// TwinCAT 3 PLC project TcoTixonFeeding
// Title: TcoTixonFeeding
// Company: Vortex.Library
// Author: TcOpenGroup
// ProjectVersion: 0.6.0.913
// ProgramVersion: 3.1.4024.12
// libraries:
//   Tc2_Standard, * (Beckhoff Automation GmbH)
//   Tc2_System, * (Beckhoff Automation GmbH)
//   Tc3_Module, * (Beckhoff Automation GmbH)
//   TcoAbstractions, 0.6.0.913 (Vortex.Library)
//   TcoCore, 0.6.0.913 (Vortex.Library)
//   TcoIo, 0.6.0.913 (Vortex.Library)
//   TcoUtilities, 0.6.0.913 (Vortex.Library)
// project tree:
//   DUTs/ TcoTixonGenericConfig.TcDUT, TcoTixonGenericPickConfig.TcDUT, TcoTixonGenericControl.TcDUT, TcoTixonGenericStatus.TcDUT
//   DUTs/TixonPickStep/ TcoTixonPickStep_Config_v_1_x_x.TcDUT, TcoTixonPickStep_Control_v_1_x_x.TcDUT, TcoTixonPickStep_Status_v_1_x_x.TcDUT
//   DUTs/TixonPickVibroBasic/ TcoTixonPickVibroBasic_Config_v_1_x_x.TcDUT, TcoTixonPickVibroBasic_Control_v_1_x_x.TcDUT, TcoTixonPickVibroBasic_Status_v_1_x_x.TcDUT
//   DUTs/TixonStep/ TcoTixonStep_Config_v_1_x_x.TcDUT, TcoTixonStep_Control_v_1_x_x.TcDUT, TcoTixonStep_Status_v_1_x_x.TcDUT
//   DUTs/TixonVibro/ TcoTixonVibro_Config_v_1_x_x.TcDUT, TcoTixonVibro_Control_v_1_x_x.TcDUT, TcoTixonVibro_Status_v_1_x_x.TcDUT
//   DUTs/TixonPickVibro/ TcoTixonPickVibro_Config_v_1_x_x.TcDUT, TcoTixonPickVibro_Control_v_1_x_x.TcDUT, TcoTixonPickVibro_Status_v_1_x_x.TcDUT
//   / PlcTask.TcTTO
//   POUs/ MAIN.TcPOU
//   POUs/Prototypes/GenericTasks/Base/ TcoTixonFeedingTask.TcPOU
//   POUs/Prototypes/GenericTasks/Buffer/ TcoTixonBufferTask.TcPOU, TcoTixonPickBufferTask.TcPOU
//   POUs/Prototypes/GenericTasks/Hopper/ TcoTixonHopperTask.TcPOU
//   POUs/Prototypes/TiconPickStep/Taks/Step/ TcoTixonPickStepTask.TcPOU
//   POUs/Prototypes/TiconPickStep/Taks/ TcoTixonPickStepSeparatorTask.TcPOU
//   POUs/Prototypes/TiconPickStep/ TcoTixonPickStep_v_1_x_x.TcPOU
//   POUs/Prototypes/TiconPickVibro/Taks/ TcoTixonPickVibroFeederTask.TcPOU, TcoTixonPickVibroSeparatorTask.TcPOU
//   POUs/Prototypes/TiconPickVibro/ TcoTixonPickVibro_v_1_x_x.TcPOU
//   POUs/Prototypes/TixonPickVibroBasic/Tasks/ TcoTixonPickVibroBasicSeparatorTask.TcPOU
//   POUs/Prototypes/TixonPickVibroBasic/ TcoTixonPickVibroBasic_v_1_x_x.TcPOU
//   POUs/Prototypes/TixonStep/Tasks/Separe/ TcoTixonStepSeparatorTask.TcPOU
//   POUs/Prototypes/TixonStep/Tasks/Step/ TcoTixonStepTask.TcPOU
//   POUs/Prototypes/TixonStep/ TcoTixonStep_v_1_x_x.TcPOU
//   POUs/Prototypes/TixonVibro/Tasks/Separe/ TcoTixonVibroSeparatorTask.TcPOU
//   POUs/Prototypes/TixonVibro/ TcoTixonVibro_v_1_x_x.TcPOU
// real-time tasks:
//   TASK PlcTask: cycle T#10ms, priority 20, ADS port 350
//   TASK PlcTask1: cycle T#10ms, priority 1, ADS port 351
//   TASK PN: cycle T#8ms, priority 2, ADS port 301
// I/O:
//   DEVICE Device 4 (EtherCAT) (disabled), AmsNetId 172.20.10.104.5.1
//     Term 1 (EK1100) [EK1100 EtherCAT Coupler (2A E-Bus)]
//       Term 2 (EL1008) [EL1008 8Ch. Dig. Input 24V, 3ms]
//       Term 3 (EL2008) [EL2008 8Ch. Dig. Output 24V, 0.5A]
//       Term 4 (EL3052) [EL3052 2Ch. Ana. Input 4-20mA]
//       Term 5 (EL9576) [EL9576 Brake chopper terminal]
//       Term 6 (EL7211-0010) [EL7211-0010 1Ch. MDP742 Servo motor output stage with OCT (50V, 4.5A RMS)]
//       Term 14 (EL7047) [EL7047 1Ch. Stepper motor output stage (50V, 5A)]
//       Term 8 (EL9011) [EL9011 End Terminal]
//   DEVICE Device 1 (EtherCAT) (disabled), AmsNetId 192.168.4.1.2.1
//     Drive 7 (IndraDrive MPB20) [IndraDrive MPB20]
//   DEVICE ECAT (disabled), AmsNetId 192.168.4.1.3.1
//     EK1200 [EK1200-5000 EtherCAT Power supply (2A E-Bus)]
//       IA1 [EL1008 8Ch. Dig. Input 24V, 3ms]
//       QA1 [EL2008 8Ch. Dig. Output 24V, 0.5A]
//       Term 4 (EL9011) [EL9011 End Terminal]
// variable links:
//   TcoTixonFeedingTests/TcoTixonFeedingTests Instance <-> ECAT
//     PlcTask1 Inputs/GVL_iXlinker.ECAT_x.InfoData.AmsNetId <-> InfoData/AmsNetId
//     PlcTask1 Inputs/GVL_iXlinker.ECAT_x.InfoData.CfgSlaveCount <-> InfoData/CfgSlaveCount
//     PlcTask1 Inputs/GVL_iXlinker.ECAT_x.InfoData.ChangeCount <-> InfoData/ChangeCount
//     PlcTask1 Inputs/GVL_iXlinker.ECAT_x.InfoData.DevId <-> InfoData/DevId
//     PlcTask1 Inputs/GVL_iXlinker.ECAT_x.Inputs.DevState <-> Inputs/DevState
//     PlcTask1 Inputs/GVL_iXlinker.ECAT_x.Inputs.Frm0InputToggle <-> Inputs/Frm0InputToggle
//     PlcTask1 Inputs/GVL_iXlinker.ECAT_x.Inputs.Frm0State <-> Inputs/Frm0State
//     PlcTask1 Inputs/GVL_iXlinker.ECAT_x.Inputs.Frm0WcState <-> Inputs/Frm0WcState
//     PlcTask1 Inputs/GVL_iXlinker.ECAT_x.Inputs.SlaveCount <-> Inputs/SlaveCount
//     PlcTask1 Outputs/GVL_iXlinker.ECAT_x.Outputs.DevCtrl <-> Outputs/DevCtrl
//     PlcTask1 Outputs/GVL_iXlinker.ECAT_x.Outputs.Frm0Ctrl <-> Outputs/Frm0Ctrl
//     PlcTask1 Outputs/GVL_iXlinker.ECAT_x.Outputs.Frm0WcCtrl <-> Outputs/Frm0WcCtrl
//   TcoTixonFeedingTests/TcoTixonFeedingTests Instance <-> ECAT/EK1200/IA1
//     PlcTask1 Inputs/GVL_iXlinker.ECAT_x.EK1200.IA1.Channel_{1..8}.Input <-> Channel {1..8}/Input  (8 links)
//     PlcTask1 Inputs/GVL_iXlinker.ECAT_x.EK1200.IA1.InfoData.State <-> InfoData/State
//     PlcTask1 Inputs/GVL_iXlinker.ECAT_x.EK1200.IA1.WcState.InputToggle <-> WcState/InputToggle
//     PlcTask1 Inputs/GVL_iXlinker.ECAT_x.EK1200.IA1.WcState.WcState <-> WcState/WcState
//   TcoTixonFeedingTests/TcoTixonFeedingTests Instance <-> ECAT/EK1200/QA1
//     PlcTask1 Inputs/GVL_iXlinker.ECAT_x.EK1200.QA1.InfoData.State <-> InfoData/State
//     PlcTask1 Inputs/GVL_iXlinker.ECAT_x.EK1200.QA1.WcState.WcState <-> WcState/WcState
//     PlcTask1 Outputs/GVL_iXlinker.ECAT_x.EK1200.QA1.Channel_{1..8}.Output <-> Channel {1..8}/Output  (8 links)

CONFIGURATION TcoTixonFeeding
    RESOURCE PLC ON TwinCAT3
        TASK PlcTask(INTERVAL := T#10ms, PRIORITY := 20);
        PROGRAM MAIN WITH PlcTask : MAIN;
    END_RESOURCE
END_CONFIGURATION

// ---- DUTs/TcoTixonGenericConfig.TcDUT
TYPE TcoTixonGenericConfig :
STRUCT
    {attribute addProperty Name "<#Blink period#> - T_BLINK"}
    BlinkTime : TIME := T#500MS;
    {attribute addProperty Name "<#Feeder empty time to report#> - T_SIG_EMPTY"}
    FeederEmptyTime : TIME := T#5S;
    {attribute addProperty Name "<#Buffer empty time to report#> - T_BUF_EMPTY"}
    BufferEmptyTime : TIME := T#1S;
    {attribute addProperty Name "<#Buffer full time to report#> - T_BUF_FULL"}
    BufferFullTime : TIME := T#1S;
    {attribute addProperty Name "<#Buffer blow on start#> - T_BUF_BLOW_ON"}
    BufferBlowStartTime : TIME := T#300MS;
    {attribute addProperty Name "<#Buffer time to idle#> - T_BUF_IDLE"}
    BufferIdleTime : TIME := T#5S;
    {attribute addProperty Name "<#Buffer full blow time after#> - T_BUF_BLOW_FULL"}
    BufferBlowFullTime : TIME := T#1S;
    {attribute addProperty Name "<#Buffer blow  active #>"}
    BufferBlowActive : BOOL := TRUE;
    {attribute addProperty Name "<#Time when component in separator #> - T_BUFSEP_ON"}
    TimeToComponentInSeparator : TIME := T#300MS;
    {attribute addProperty Name "<#Time when component is out of separator #> - T_FLY_OFF"}
    TimeToComponentOutSeparator : TIME := T#1S;
    {attribute addProperty Name "<#Hooper is active#>"}
    HopperActive : BOOL := FALSE;
    {attribute addProperty Name "<#Time to hopper start #> - T_HOOP_ON"}
    TimeToHopperStart : TIME := T#5S;
    {attribute addProperty Name "<#Time to hopper run #> - T_HOOP_RUN"}
    TimeToHopperRun : TIME := T#30S;
END_STRUCT
END_TYPE

// ---- DUTs/TcoTixonGenericPickConfig.TcDUT
TYPE TcoTixonGenericPickConfig EXTENDS TcoTixonGenericConfig :
STRUCT
    {attribute addProperty Name "<#Separator  active #>"}
    SeparatorActive : BOOL := TRUE;
END_STRUCT
END_TYPE

// ---- DUTs/TcoTixonGenericControl.TcDUT
TYPE TcoTixonGenericControl :
STRUCT
    {attribute addProperty Name "<#Feeding A #> - q1"}
    FeedingA : BOOL;
    {attribute addProperty Name "<#Separe component#> - q2"}
    SepareComponent : BOOL;
    {attribute addProperty Name "<#Blow A#> - q3"}
    BlowAValve : BOOL;
    {attribute addProperty Name "<#Red led#> - q4"}
    RedLed : BOOL;
    {attribute addProperty Name "<#Green led#> - q5"}
    GreenLed : BOOL;
    {attribute addProperty Name "<#Hooper#> - q6"}
    Hooper : BOOL;
END_STRUCT
END_TYPE

// ---- DUTs/TcoTixonGenericStatus.TcDUT
TYPE TcoTixonGenericStatus :
STRUCT
    ActionDescription : STRING(100);
    {attribute addProperty Name "<#Component is ready#>"}
    ComponentReady : BOOL;
    {attribute addProperty Name "<#Tixon controller in auto#> - i1"}
    ControllerInAuto : BOOL;
    {attribute addProperty Name "<#Feeder has components#> - i2"}
    NotEmptyFeeder : BOOL;
    {attribute addProperty Name "<#Separator in home position#> - i3"}
    SeparatorHomePos : BOOL;
    {attribute addProperty Name "<#Filing sensor#> - i4"}
    FillingSensor : BOOL;
    {attribute addProperty Name "<#Separator present#> - i5"}
    SeparatorPresent : BOOL;
END_STRUCT
END_TYPE

// ---- DUTs/TixonPickStep/TcoTixonPickStep_Config_v_1_x_x.TcDUT
TYPE TcoTixonPickStep_Config_v_1_x_x EXTENDS TcoTixonGenericPickConfig :
STRUCT
    {attribute addProperty Name "<#Time when stepper in work #> - T_STEP_WORK"}
    SteperInWorkTime : TIME := T#1S;
    {attribute addProperty Name "<#Time when stepper in home #> - T_STEP_HOME"}
    SteperInHomeTime : TIME := T#1S;
    {attribute addProperty Name "<#Error time separator #> - T_SEP_ERROR"}
    ErrorTimeSeparator : TIME := T#0S;
    {attribute addProperty Name "<#Error time buffer #> - T_BUFF_ERROR"}
    ErrorTimeBuffer : TIME := T#0S;
    {attribute addProperty Name "<#Error time Stepper #> - T_STEP_ERROR"}
    ErrorTimeStepper : TIME := T#0S;
    {attribute addProperty Name "<#Error time Hopper #> - T_HOP_ERROR"}
    ErrorTimeHopper : TIME := T#0S;
END_STRUCT
END_TYPE

// ---- DUTs/TixonPickStep/TcoTixonPickStep_Control_v_1_x_x.TcDUT
TYPE TcoTixonPickStep_Control_v_1_x_x EXTENDS TcoTixonGenericControl :
STRUCT
    {attribute addProperty Name "<#Stepper valve#> - q7"}
    StepperValve : BOOL;
END_STRUCT
END_TYPE

// ---- DUTs/TixonPickStep/TcoTixonPickStep_Status_v_1_x_x.TcDUT
TYPE TcoTixonPickStep_Status_v_1_x_x EXTENDS TcoTixonGenericStatus :
STRUCT
    {attribute addProperty Name "<#Separator in work position#> - i6"}
    SeparatorWorkPos : BOOL;
    {attribute addProperty Name "<#Stepper in home position#> - i7 "}
    StepperHomePos : BOOL;
    {attribute addProperty Name "<#Stepper in work position#> - i8"}
    StepperWorkPos : BOOL;
    {attribute addProperty Name "<#In Pick Zone#>"}
    InPickZone : BOOL;
END_STRUCT
END_TYPE

// ---- DUTs/TixonPickVibroBasic/TcoTixonPickVibroBasic_Config_v_1_x_x.TcDUT
TYPE TcoTixonPickVibroBasic_Config_v_1_x_x EXTENDS TcoTixonGenericPickConfig :
STRUCT
    {attribute addProperty Name "<#Error time separator #> - T_SEP_ERROR"}
    ErrorTimeSeparator : TIME := T#0S;
    {attribute addProperty Name "<#Error time buffer #> - T_BUFF_ERROR"}
    ErrorTimeBuffer : TIME := T#0S;
    {attribute addProperty Name "<#Error time Hopper #> - T_HOP_ERROR"}
    ErrorTimeHopper : TIME := T#0S;
END_STRUCT
END_TYPE

// ---- DUTs/TixonPickVibroBasic/TcoTixonPickVibroBasic_Control_v_1_x_x.TcDUT
TYPE TcoTixonPickVibroBasic_Control_v_1_x_x EXTENDS TcoTixonGenericControl :
STRUCT
END_STRUCT
END_TYPE

// ---- DUTs/TixonPickVibroBasic/TcoTixonPickVibroBasic_Status_v_1_x_x.TcDUT
TYPE TcoTixonPickVibroBasic_Status_v_1_x_x EXTENDS TcoTixonGenericStatus :
STRUCT
    {attribute addProperty Name "<#Separator in work position#> - i6"}
    SeparatorWorkPos : BOOL;
    {attribute addProperty Name "<#In Pick Zone#>"}
    InPickZone : BOOL;
END_STRUCT
END_TYPE

// ---- DUTs/TixonStep/TcoTixonStep_Config_v_1_x_x.TcDUT
TYPE TcoTixonStep_Config_v_1_x_x EXTENDS TcoTixonGenericConfig :
STRUCT
    {attribute addProperty Name "<#Time when stepper in work #> - T_STEP_WORK"}
    SteperInWorkTime : TIME := T#1S;
    {attribute addProperty Name "<#Time when stepper in home #> - T_STEP_HOME"}
    SteperInHomeTime : TIME := T#1S;
    {attribute addProperty Name "<#Error time separator #> - T_SEP_ERROR"}
    ErrorTimeSeparator : TIME := T#0S;
    {attribute addProperty Name "<#Error time buffer #> - T_BUFF_ERROR"}
    ErrorTimeBuffer : TIME := T#0S;
    {attribute addProperty Name "<#Error time Stepper #> - T_STEP_ERROR"}
    ErrorTimeStepper : TIME := T#0S;
    {attribute addProperty Name "<#Error time Hopper #> - T_HOP_ERROR"}
    ErrorTimeHopper : TIME := T#0S;
    {attribute addProperty Name "<#Out of box sensor disabled (usualy TRUE when pushing to up direction) #>"}
    OutOfBoxSensorDisabled : BOOL := FALSE;
    {attribute addProperty Name "<#Separator has work position (usualy TRUE when pushing to up direction)#>"}
    SeparatorHasWorkPosition : BOOL := FALSE;
    {attribute addProperty Name "<#Buffer stucked on filing sensor#> - T_BUF_STUCK_FIL_SENSOR"}
    BufferStuckedOnFillingSensor : TIME := T#20S;
END_STRUCT
END_TYPE

// ---- DUTs/TixonStep/TcoTixonStep_Control_v_1_x_x.TcDUT
TYPE TcoTixonStep_Control_v_1_x_x EXTENDS TcoTixonGenericControl :
STRUCT
    {attribute addProperty Name "<#Stepper valve#> - q7"}
    StepperValve : BOOL;
    {attribute addProperty Name "<#Shot component#> - q8"}
    ShotComponent : BOOL;
END_STRUCT
END_TYPE

// ---- DUTs/TixonStep/TcoTixonStep_Status_v_1_x_x.TcDUT
TYPE TcoTixonStep_Status_v_1_x_x EXTENDS TcoTixonGenericStatus :
STRUCT
    {attribute addProperty Name "<#Stepper in home position#> - i6 "}
    StepperHomePos : BOOL;
    {attribute addProperty Name "<#Stepper in work position#> - i7"}
    StepperWorkPos : BOOL;
    {attribute addProperty Name "<#Component out of box#> - i8"}
    ComponentOutOfBox : BOOL;
    {attribute addProperty Name "<#Separator in work position#> - i9"}
    SeparatorWorkPos : BOOL;
END_STRUCT
END_TYPE

// ---- DUTs/TixonVibro/TcoTixonVibro_Config_v_1_x_x.TcDUT
TYPE TcoTixonVibro_Config_v_1_x_x EXTENDS TcoTixonGenericConfig :
STRUCT
    {attribute addProperty Name "<#Error time separator #> - T_SEP_ERROR"}
    ErrorTimeSeparator : TIME := T#0S;
    {attribute addProperty Name "<#Error time buffer #> - T_BUFF_ERROR"}
    ErrorTimeBuffer : TIME := T#0S;
    {attribute addProperty Name "<#Error time Hopper #> - T_HOP_ERROR"}
    ErrorTimeHopper : TIME := T#0S;
    {attribute addProperty Name "<#Out of box sensor disabled (usualy TRUE when pushing to up direction) #>"}
    OutOfBoxSensorDisabled : BOOL := FALSE;
    {attribute addProperty Name "<#Separator has work position (usualy TRUE when pushing to up direction)#>"}
    SeparatorHasWorkPosition : BOOL := FALSE;
END_STRUCT
END_TYPE

// ---- DUTs/TixonVibro/TcoTixonVibro_Control_v_1_x_x.TcDUT
TYPE TcoTixonVibro_Control_v_1_x_x EXTENDS TcoTixonGenericControl :
STRUCT
    {attribute addProperty Name "<#Shot component#> - q7"}
    ShotComponent : BOOL;
END_STRUCT
END_TYPE

// ---- DUTs/TixonVibro/TcoTixonVibro_Status_v_1_x_x.TcDUT
TYPE TcoTixonVibro_Status_v_1_x_x EXTENDS TcoTixonGenericStatus :
STRUCT
    {attribute addProperty Name "<#Component out of box#>- i6"}
    ComponentOutOfBox : BOOL;
    {attribute addProperty Name "<#Separator in work position#> - i7"}
    SeparatorWorkPos : BOOL;
END_STRUCT
END_TYPE

// ---- DUTs/TixonPickVibro/TcoTixonPickVibro_Config_v_1_x_x.TcDUT
TYPE TcoTixonPickVibro_Config_v_1_x_x EXTENDS TcoTixonGenericPickConfig :
STRUCT
    {attribute addProperty Name "<#Feeder blow B on start#> - T_FEEDER_BLOWB_ON"}
    FeederBlowBStartTime : TIME := T#300MS;
    {attribute addProperty Name "<#Feeder full blow B time after#> - T_FEEDER_BLOWB_FULL"}
    FeederBlowBFullTime : TIME := T#1S;
    {attribute addProperty Name "<#Feeder blow B  active #>"}
    FeederBlowBActive : BOOL := FALSE;
    {attribute addProperty Name "<#Error time separator #> - T_SEP_ERROR"}
    ErrorTimeSeparator : TIME := T#0S;
    {attribute addProperty Name "<#Error time buffer #> - T_BUFF_ERROR"}
    ErrorTimeBuffer : TIME := T#0S;
    {attribute addProperty Name "<#Error time Hopper #> - T_HOP_ERROR"}
    ErrorTimeHopper : TIME := T#0S;
END_STRUCT
END_TYPE

// ---- DUTs/TixonPickVibro/TcoTixonPickVibro_Control_v_1_x_x.TcDUT
TYPE TcoTixonPickVibro_Control_v_1_x_x EXTENDS TcoTixonGenericControl :
STRUCT
    {attribute addProperty Name "<#Feeding B#> - q7 "}
    FeedingB : BOOL;
    {attribute addProperty Name "<#Blow B#> - q8"}
    BlowValveB : BOOL;
END_STRUCT
END_TYPE

// ---- DUTs/TixonPickVibro/TcoTixonPickVibro_Status_v_1_x_x.TcDUT
TYPE TcoTixonPickVibro_Status_v_1_x_x EXTENDS TcoTixonGenericStatus :
STRUCT
    {attribute addProperty Name "<#Separator in work position#> - i6"}
    SeparatorWorkPos : BOOL;
    {attribute addProperty Name "<#In Pick Zone#>"}
    InPickZone : BOOL;
END_STRUCT
END_TYPE

// ---- POUs/MAIN.TcPOU
PROGRAM MAIN
VAR
END_VAR

END_PROGRAM

// ---- POUs/Prototypes/GenericTasks/Base/TcoTixonFeedingTask.TcPOU
FUNCTION_BLOCK PUBLIC ABSTRACT TcoTixonFeedingTask EXTENDS TcoCore.TcoTask
VAR
    _errorMessage : TcoCore.TcoMessenger(THIS^);
    {attribute 'hide'}
    _progress : INT := 0;
    {attribute 'hide'}
    _infoTimer : TON;
    _infoTime : TIME;
    {attribute 'hide'}
    _errorTimer : TON;
    _errorTime : TIME;
    {attribute 'hide'}
    _timer : TON;
    {attribute 'hide'}
    _varInfo : __SYSTEM.VAR_INFO;
    {attribute 'hide'}
    _sb : TcoCore.StringBuilder;
    {attribute 'hide'}
    _autoRestore : BOOL;
END_VAR

PROPERTY PUBLIC AutoRestore : BOOL
GET
AutoRestore := _autoRestore;
END_GET
SET
_autoRestore := AutoRestore;
END_SET
END_PROPERTY

METHOD CallTimers
VAR_INPUT
    inValue : BOOL;
END_VAR
IF THIS^.ErrorTime <> T#0S OR NOT inValue THEN
    _errorTimer(IN := inValue, PT := THIS^.ErrorTime);
END_IF;

IF THIS^.InfoTime <> T#0S OR NOT inValue THEN
    _infoTimer(IN := inValue, PT := THIS^.InfoTime);
END_IF;
END_METHOD

PROPERTY PUBLIC ErrorTime : REFERENCE TO TIME
GET
ErrorTime REF= _errorTime;
END_GET
END_PROPERTY

PROPERTY InfoTime : REFERENCE TO TIME
GET
InfoTime REF= _infoTime;
END_GET
END_PROPERTY

(*~
    <docu>
        <summary>
            Restores this instance to the Ready state. Can be called explicitly or from within one of the restore mechanisms.
            <para>
                See also <see cref="PlcDocu.TcoCore.TcoTask.AutoRestorable()"/>
            </para>
        </summary>
    </docu>
~*)
METHOD Restore : ITcoRestorable
SUPER^.Restore();
_progress := 0;
_timer(In := FALSE);
CallTimers(FALSE);
Messenger.UnPin();
_errorMessage.UnPin();
_autoRestore := false;
END_METHOD

END_FUNCTION_BLOCK

// ---- POUs/Prototypes/GenericTasks/Buffer/TcoTixonBufferTask.TcPOU
FUNCTION_BLOCK TcoTixonBufferTask EXTENDS TcoTixonFeedingTask
VAR_IN_OUT
    inoConfig : TcoTixonGenericConfig;
    inoControl : TcoTixonGenericControl;
    inoStatus : TcoTixonGenericStatus;
END_VAR

IF Execute() THEN
    IF _progress = 0 THEN
        IF NOT __ISVALIDREF(inoControl) THEN
            _varInfo := __VARINFO(inoControl);
            Messenger.Programming(_sb.Clear().Append('<#Invalid reference: #>').Append(_varInfo.Symbol).ToString()).Pin();
        ELSIF NOT __ISVALIDREF(inoConfig) THEN
            _varInfo := __VARINFO(inoConfig);
            Messenger.Programming(_sb.Clear().Append('<#Invalid reference: #>').Append(_varInfo.Symbol).ToString()).Pin();
        ELSIF NOT __ISVALIDREF(inoStatus) THEN
            _varInfo := __VARINFO(inoStatus);
            Messenger.Programming(_sb.Clear().Append('<#Invalid reference: #>').Append(_varInfo.Symbol).ToString()).Pin();
        ELSIF NOT inoStatus.ControllerInAuto THEN
            _varInfo := __VARINFO(inoStatus.ControllerInAuto);
            Messenger.Warning(_sb.Clear().Append('<#Tixon control system not in auto #>').Append(_varInfo.Symbol).ToString());
        ELSE
            IF NOT THIS^._errorMessage.Pinned THEN
                _progress := _progress + 1;
            END_IF;
        END_IF
    END_IF

    IF _progress = 1 THEN
        Messenger.Debug('<#Waiting for buffer is Empty #>');

        _timer(IN := NOT inoStatus.FillingSensor OR (inoStatus.SeparatorHomePos AND NOT inoStatus.SeparatorPresent),
            Pt := inoConfig.BufferEmptyTime);

        IF _timer.Q THEN
            _progress := _progress + 1;
            _timer(In := FALSE);
        END_IF;
    END_IF;

    IF _progress = 2 THEN
        Messenger.Debug('<#Waiting for blow on #>');
        _timer(IN := TRUE, Pt := inoConfig.BufferBlowStartTime);
        inoControl.BlowAValve := inoConfig.BufferBlowActive;

        IF _timer.Q OR NOT inoConfig.BufferBlowActive THEN
            inoControl.FeedingA := TRUE;
            _progress := _progress + 1;
            _timer(In := FALSE);
        END_IF;
    END_IF;

    IF _progress = 3 THEN
        Messenger.Debug('<#Waiting for buffer is full and go idle#>');
        _timer(IN := inoStatus.FillingSensor AND InoStatus.SeparatorPresent, Pt := inoConfig.BufferIdleTime);

        IF _timer.Q THEN
            _progress := _progress + 1;
            _timer(In := FALSE);
        END_IF
    END_IF;

    IF _progress = 4 THEN
        inoControl.FeedingA := FALSE;
        Messenger.Debug('<#Waiting for buffer is full and blow ending#>');
        _timer(IN := TRUE, Pt := inoConfig.BufferBlowFullTime);

        IF _timer.Q OR NOT inoConfig.BufferBlowActive THEN
            inoControl.BlowAValve := FALSE;
            _progress := _progress + 1;
            _timer(In := FALSE);
        END_IF;
    END_IF;

    IF _progress = 5 THEN
        THIS^.DoneWhen(TRUE);
    END_IF;

    CallTimers(_progress > 1); //empty and start feeding
    THIS^.ThrowWhen(_errorTimer.Q);
END_IF

IF THIS^.Error AND NOT _errorMessage.Pinned THEN
    THIS^.Restore();
END_IF

(*~
    <docu>
        <summary>
            Executes when task is aborted.
        </summary>
    </docu>
~*)
METHOD PROTECTED OnAbort
IF __ISVALIDREF(inoStatus) THEN
    THIS^.inoStatus.ActionDescription := '<#Buffer task  was aborted.#>';
END_IF;
END_METHOD

(*~
    <docu>
        <summary>
            Executes when task reaches the ```Done``` state .
        </summary>
    </docu>
~*)
METHOD PROTECTED OnDone
IF __ISVALIDREF(inoStatus) THEN
    THIS^.inoStatus.ActionDescription := '<#Buffer task  finished successfully.#>';
END_IF;

_progress := 0;

IF AutoRestore THEN
    Restore();
END_IF
END_METHOD

METHOD PROTECTED OnError
VAR
    description : STRING;
END_VAR
description := '<#Buffer task finished with error.#>';
inoControl.FeedingA := FALSE;
inoControl.BlowAValve := false;

IF __ISVALIDREF(inoStatus) THEN
    THIS^.inoStatus.ActionDescription := description;
END_IF;

THIS^._errorMessage.Error(_sb.Clear().Append(description).Append(' To restore acknowledge this alarm.').ToString()).Pin();
END_METHOD

METHOD PROTECTED OnStart
IF __ISVALIDREF(inoStatus) THEN
    THIS^.inoStatus.ActionDescription := '<#Buffer task started.#>';
END_IF;

CallTimers(FALSE);
END_METHOD

(*~
    <docu>
        <summary>
            Restores this instance to the Ready state. Can be called explicitly or from within one of the restore mechanisms.
            <para>
                See also <see cref="PlcDocu.TcoCore.TcoTask.AutoRestorable()"/>
            </para>
        </summary>
    </docu>
~*)
METHOD Restore : ITcoRestorable
SUPER^.Restore();
END_METHOD

END_FUNCTION_BLOCK

// ---- POUs/Prototypes/GenericTasks/Buffer/TcoTixonPickBufferTask.TcPOU
FUNCTION_BLOCK TcoTixonPickBufferTask EXTENDS TcoTixonFeedingTask
VAR_IN_OUT
    inoConfig : TcoTixonGenericPickConfig;
    inoControl : TcoTixonGenericControl;
    inoStatus : TcoTixonGenericStatus;
END_VAR

IF Execute() THEN
    IF _progress = 0 THEN
        IF NOT __ISVALIDREF(inoControl) THEN
            _varInfo := __VARINFO(inoControl);
            Messenger.Programming(_sb.Clear().Append('<#Invalid reference: #>').Append(_varInfo.Symbol).ToString()).Pin();
        ELSIF NOT __ISVALIDREF(inoConfig) THEN
            _varInfo := __VARINFO(inoConfig);
            Messenger.Programming(_sb.Clear().Append('<#Invalid reference: #>').Append(_varInfo.Symbol).ToString()).Pin();
        ELSIF NOT __ISVALIDREF(inoStatus) THEN
            _varInfo := __VARINFO(inoStatus);
            Messenger.Programming(_sb.Clear().Append('<#Invalid reference: #>').Append(_varInfo.Symbol).ToString()).Pin();
        ELSIF NOT inoStatus.ControllerInAuto THEN
            _varInfo := __VARINFO(inoStatus.ControllerInAuto);
            Messenger.Warning(_sb.Clear().Append('<#Tixon control system not in auto #>').Append(_varInfo.Symbol).ToString());
        ELSE
            IF NOT THIS^._errorMessage.Pinned THEN
                _progress := _progress + 1;
            END_IF;
        END_IF
    END_IF

    IF _progress = 1 THEN
        Messenger.Debug('<#Waiting for buffer is Empty #>');
        _timer(IN := NOT inoStatus.FillingSensor OR (NOT inoStatus.SeparatorPresent), Pt := inoConfig.BufferEmptyTime);

        IF _timer.Q THEN
            _progress := _progress + 1;
            _timer(In := FALSE);
        END_IF;
    END_IF;

    IF _progress = 2 THEN
        Messenger.Debug('<#Waiting for blow on #>');
        _timer(IN := TRUE, Pt := inoConfig.BufferBlowStartTime);
        inoControl.BlowAValve := inoConfig.BufferBlowActive;

        IF _timer.Q OR NOT inoConfig.BufferBlowActive THEN
            inoControl.FeedingA := TRUE;
            _progress := _progress + 1;
            _timer(In := FALSE);
        END_IF;
    END_IF;

    IF _progress = 3 THEN
        Messenger.Debug('<#Waiting for buffer is full and go idle#>');
        _timer(IN := inoStatus.FillingSensor AND InoStatus.SeparatorPresent, Pt := inoConfig.BufferIdleTime);

        IF _timer.Q THEN
            _progress := _progress + 1;
            _timer(In := FALSE);
        END_IF
    END_IF;

    IF _progress = 4 THEN
        inoControl.FeedingA := FALSE;
        Messenger.Debug('<#Waiting for buffer is full and blow ending#>');
        _timer(IN := TRUE, Pt := inoConfig.BufferBlowFullTime);

        IF _timer.Q OR NOT inoConfig.BufferBlowActive THEN
            inoControl.BlowAValve := FALSE;
            _progress := _progress + 1;
            _timer(In := FALSE);
        END_IF;
    END_IF;

    IF _progress = 5 THEN
        THIS^.DoneWhen(TRUE);
    END_IF;

    CallTimers(_progress > 1); //empty and start feeding
    THIS^.ThrowWhen(_errorTimer.Q);
END_IF

IF THIS^.Error AND NOT _errorMessage.Pinned THEN
    THIS^.Restore();
END_IF

(*~
    <docu>
        <summary>
            Executes when task is aborted.
        </summary>
    </docu>
~*)
METHOD PROTECTED OnAbort
IF __ISVALIDREF(inoStatus) THEN
    THIS^.inoStatus.ActionDescription := '<#Buffer task  was aborted.#>';
END_IF;
END_METHOD

(*~
    <docu>
        <summary>
            Executes when task reaches the ```Done``` state .
        </summary>
    </docu>
~*)
METHOD PROTECTED OnDone
IF __ISVALIDREF(inoStatus) THEN
    THIS^.inoStatus.ActionDescription := '<#Buffer task  finished successfully.#>';
END_IF;

_progress := 0;

IF AutoRestore THEN
    Restore();
END_IF
END_METHOD

METHOD PROTECTED OnError
VAR
    description : STRING;
END_VAR
description := '<#Buffer task finished with error.#>';
inoControl.FeedingA := FALSE;
inoControl.BlowAValve := false;

IF __ISVALIDREF(inoStatus) THEN
    THIS^.inoStatus.ActionDescription := description;
END_IF;

THIS^._errorMessage.Error(_sb.Clear().Append(description).Append(' To restore acknowledge this alarm.').ToString()).Pin();
END_METHOD

METHOD PROTECTED OnStart
IF __ISVALIDREF(inoStatus) THEN
    THIS^.inoStatus.ActionDescription := '<#Buffer task started.#>';
END_IF;

CallTimers(FALSE);
END_METHOD

(*~
    <docu>
        <summary>
            Restores this instance to the Ready state. Can be called explicitly or from within one of the restore mechanisms.
            <para>
                See also <see cref="PlcDocu.TcoCore.TcoTask.AutoRestorable()"/>
            </para>
        </summary>
    </docu>
~*)
METHOD Restore : ITcoRestorable
SUPER^.Restore();
END_METHOD

END_FUNCTION_BLOCK

// ---- POUs/Prototypes/GenericTasks/Hopper/TcoTixonHopperTask.TcPOU
FUNCTION_BLOCK TcoTixonHopperTask EXTENDS TcoTixonFeedingTask
VAR_IN_OUT
    inoConfig : TcoTixonGenericConfig;
    inoControl : TcoTixonGenericControl;
    inoStatus : TcoTixonGenericStatus;
END_VAR

IF Execute() THEN
    IF _progress = 0 THEN
        IF NOT __ISVALIDREF(inoControl) THEN
            _varInfo := __VARINFO(inoControl);
            Messenger.Programming(_sb.Clear().Append('<#Invalid reference: #>').Append(_varInfo.Symbol).ToString()).Pin();
        ELSIF NOT __ISVALIDREF(inoConfig) THEN
            _varInfo := __VARINFO(inoConfig);
            Messenger.Programming(_sb.Clear().Append('<#Invalid reference: #>').Append(_varInfo.Symbol).ToString()).Pin();
        ELSIF NOT __ISVALIDREF(inoStatus) THEN
            _varInfo := __VARINFO(inoStatus);
            Messenger.Programming(_sb.Clear().Append('<#Invalid reference: #>').Append(_varInfo.Symbol).ToString()).Pin();
        ELSIF NOT inoStatus.ControllerInAuto THEN
            _varInfo := __VARINFO(inoStatus.ControllerInAuto);
            Messenger.Warning(_sb.Clear().Append('<#Tixon control system not in auto #>').Append(_varInfo.Symbol).ToString());
        ELSE
            IF NOT THIS^._errorMessage.Pinned THEN
                _progress := _progress + 1;
            END_IF;
        END_IF
    END_IF

    IF _progress = 1 THEN
        inoControl.Hooper := FALSE;
        _progress := _progress + 1;
        _timer(In := FALSE);
    END_IF;

    IF _progress = 2 THEN
        Messenger.Debug('<#Waiting for feeder empty#>');
        _timer(IN := NOT inoStatus.NotEmptyFeeder, Pt := inoConfig.TimeToHopperStart);

        IF _timer.Q THEN
            _progress := _progress + 1;
            _timer(In := FALSE);
            ;
        END_IF
    END_IF;

    IF _progress = 3 THEN
        inoControl.Hooper := TRUE;
        Messenger.Debug('<#Hopper is running#>');
        _timer(IN := inoStatus.NotEmptyFeeder, Pt := inoConfig.TimeToHopperRun);

        IF _timer.Q THEN
            _progress := _progress + 1;
            _timer(In := FALSE);
        END_IF
    END_IF;

    IF _progress = 4 THEN
        THIS^.DoneWhen(TRUE);
    END_IF;

    CallTimers(TRUE);
    THIS^.ThrowWhen(_errorTimer.Q);
END_IF

IF THIS^.Error AND NOT _errorMessage.Pinned THEN
    THIS^.Restore();
END_IF

(*~
    <docu>
        <summary>
            Executes when task is aborted.
        </summary>
    </docu>
~*)
METHOD PROTECTED OnAbort
IF __ISVALIDREF(inoStatus) THEN
    THIS^.inoStatus.ActionDescription := '<#Hopper task  was aborted.#>';
END_IF;
END_METHOD

(*~
    <docu>
        <summary>
            Executes when task reaches the ```Done``` state .
        </summary>
    </docu>
~*)
METHOD PROTECTED OnDone
IF __ISVALIDREF(inoStatus) THEN
    THIS^.inoStatus.ActionDescription := '<#Hopper task  finished successfully.#>';
END_IF;

_progress := 0;

IF AutoRestore THEN
    Restore();
END_IF
END_METHOD

METHOD PROTECTED OnError
VAR
    description : STRING;
END_VAR
description := '<#Hopper task finished with error.#>';
inoControl.Hooper := FALSE;

IF __ISVALIDREF(inoStatus) THEN
    THIS^.inoStatus.ActionDescription := description;
END_IF;

THIS^._errorMessage.Error(_sb.Clear().Append(description).Append(' To restore acknowledge this alarm.').ToString()).Pin();
END_METHOD

METHOD PROTECTED OnStart
IF __ISVALIDREF(inoStatus) THEN
    THIS^.inoStatus.ActionDescription := '<#Hopper task started.#>';
END_IF;

CallTimers(FALSE);
END_METHOD

(*~
    <docu>
        <summary>
            Restores this instance to the Ready state. Can be called explicitly or from within one of the restore mechanisms.
            <para>
                See also <see cref="PlcDocu.TcoCore.TcoTask.AutoRestorable()"/>
            </para>
        </summary>
    </docu>
~*)
METHOD Restore : ITcoRestorable
SUPER^.Restore();
END_METHOD

END_FUNCTION_BLOCK

// ---- POUs/Prototypes/TiconPickStep/Taks/Step/TcoTixonPickStepTask.TcPOU
FUNCTION_BLOCK TcoTixonPickStepTask EXTENDS TcoTixonFeedingTask
VAR_IN_OUT
    inoConfig : TcoTixonPickStep_Config_v_1_x_x;
    inoControl : TcoTixonPickStep_Control_v_1_x_x;
    inoStatus : TcoTixonPickStep_Status_v_1_x_x;
END_VAR
VAR
    _timerIsFull : TON;
END_VAR

IF Execute() THEN
    _timerIsFull(IN := inoStatus.FillingSensor, PT := inoConfig.BufferFullTime);

    IF _progress = 0 THEN
        IF NOT __ISVALIDREF(inoControl) THEN
            _varInfo := __VARINFO(inoControl);
            Messenger.Programming(_sb.Clear().Append('<#Invalid reference: #>').Append(_varInfo.Symbol).ToString()).Pin();
        ELSIF NOT __ISVALIDREF(inoConfig) THEN
            _varInfo := __VARINFO(inoConfig);
            Messenger.Programming(_sb.Clear().Append('<#Invalid reference: #>').Append(_varInfo.Symbol).ToString()).Pin();
        ELSIF NOT __ISVALIDREF(inoStatus) THEN
            _varInfo := __VARINFO(inoStatus);
            Messenger.Programming(_sb.Clear().Append('<#Invalid reference: #>').Append(_varInfo.Symbol).ToString()).Pin();
        ELSIF NOT inoStatus.ControllerInAuto THEN
            _varInfo := __VARINFO(inoStatus.ControllerInAuto);
            Messenger.Warning(_sb.Clear().Append('<#Tixon control system not in auto #>').Append(_varInfo.Symbol).ToString());
        ELSE
            IF NOT THIS^._errorMessage.Pinned THEN
                _progress := _progress + 1;
            END_IF;
        END_IF
    END_IF

    IF _progress = 1 THEN
        Messenger.Debug('<#Waiting for buffer empty#>');
        _timer(IN := NOT inoStatus.FillingSensor, Pt := inoConfig.BufferEmptyTime);

        IF _timer.Q AND inoControl.FeedingA THEN
            _progress := _progress + 1;
            _timer(In := FALSE);
        END_IF
    END_IF;

    IF _progress = 2 THEN
        inoControl.StepperValve := FALSE;
        Messenger.Debug('<#Stepper to home#>');
        _timer(IN := inoStatus.StepperHomePos, Pt := inoConfig.SteperInHomeTime);

        IF _timer.Q THEN
            _progress := _progress + 1;
            _timer(In := FALSE);
        END_IF
    END_IF;

    IF _progress = 3 THEN
        inoControl.StepperValve := TRUE;
        Messenger.Debug('<#Stepper to work#>');
        _timer(IN := inoStatus.StepperWorkPos, Pt := inoConfig.SteperInWorkTime);

        IF _timer.Q THEN
            _progress := _progress + 1;
            _timer(In := FALSE);
        END_IF
    END_IF;

    IF _progress = 4 THEN
        Messenger.Debug('<#Waiting for buffer full#>');

        IF _timerIsFull.Q THEN
            _progress := _progress + 1;
            _timer(In := FALSE);
        ELSE
            _progress := 2;
            _timer(In := FALSE);
        END_IF
    END_IF;

    IF _progress = 5 THEN
        THIS^.DoneWhen(TRUE);
    END_IF;

    CallTimers(_progress > 1); //empty and strat feeding
    THIS^.ThrowWhen(_errorTimer.Q);
END_IF

IF THIS^.Error AND NOT _errorMessage.Pinned THEN
    THIS^.Restore();
END_IF

(*~
    <docu>
        <summary>
            Executes when task is aborted.
        </summary>
    </docu>
~*)
METHOD PROTECTED OnAbort
IF __ISVALIDREF(inoStatus) THEN
    THIS^.inoStatus.ActionDescription := '<#Stepper task  was aborted.#>';
END_IF;
END_METHOD

(*~
    <docu>
        <summary>
            Executes when task reaches the ```Done``` state .
        </summary>
    </docu>
~*)
METHOD PROTECTED OnDone
IF __ISVALIDREF(inoStatus) THEN
    THIS^.inoStatus.ActionDescription := '<#Stepper task  finished successfully.#>';
END_IF;

_progress := 0;

IF AutoRestore THEN
    Restore();
END_IF
END_METHOD

METHOD PROTECTED OnError
VAR
    description : STRING;
END_VAR
description := '<#Stepper task finished with error.#>';
inoControl.StepperValve := false;

IF __ISVALIDREF(inoStatus) THEN
    THIS^.inoStatus.ActionDescription := description;
END_IF;

THIS^._errorMessage.Error(_sb.Clear().Append(description).Append(' To restore acknowledge this alarm.').ToString()).Pin();
END_METHOD

METHOD PROTECTED OnStart
IF __ISVALIDREF(inoStatus) THEN
    THIS^.inoStatus.ActionDescription := '<#Stepper task started.#>';
END_IF;

CallTimers(FALSE);
_timerIsFull(In := FALSE);
END_METHOD

(*~
    <docu>
        <summary>
            Restores this instance to the Ready state. Can be called explicitly or from within one of the restore mechanisms.
            <para>
                See also <see cref="PlcDocu.TcoCore.TcoTask.AutoRestorable()"/>
            </para>
        </summary>
    </docu>
~*)
METHOD Restore : ITcoRestorable
SUPER^.Restore();
_timerIsFull(In := FALSE);
END_METHOD

END_FUNCTION_BLOCK

// ---- POUs/Prototypes/TiconPickStep/Taks/TcoTixonPickStepSeparatorTask.TcPOU
FUNCTION_BLOCK TcoTixonPickStepSeparatorTask EXTENDS TcoTixonFeedingTask
VAR_IN_OUT
    inoConfig : TcoTixonPickStep_Config_v_1_x_x;
    inoControl : TcoTixonPickStep_Control_v_1_x_x;
    inoStatus : TcoTixonPickStep_Status_v_1_x_x;
END_VAR
VAR
    _componentReady : BOOL;
END_VAR

IF Execute() THEN
    IF _progress = 0 THEN
        IF NOT __ISVALIDREF(inoControl) THEN
            _varInfo := __VARINFO(inoControl);
            Messenger.Programming(_sb.Clear().Append('<#Invalid reference: #>').Append(_varInfo.Symbol).ToString()).Pin();
        ELSIF NOT __ISVALIDREF(inoConfig) THEN
            _varInfo := __VARINFO(inoConfig);
            Messenger.Programming(_sb.Clear().Append('<#Invalid reference: #>').Append(_varInfo.Symbol).ToString()).Pin();
        ELSIF NOT __ISVALIDREF(inoStatus) THEN
            _varInfo := __VARINFO(inoStatus);
            Messenger.Programming(_sb.Clear().Append('<#Invalid reference: #>').Append(_varInfo.Symbol).ToString()).Pin();
        ELSIF NOT inoStatus.ControllerInAuto THEN
            _varInfo := __VARINFO(inoStatus.ControllerInAuto);
            Messenger.Warning(_sb.Clear().Append('<#Tixon control system not in auto #>').Append(_varInfo.Symbol).ToString());
        ELSIF NOT inoConfig.SeparatorActive THEN
            _progress := 4;
        ELSE
            _progress := _progress + 1;
        END_IF
    END_IF

    IF _progress = 1 THEN
        inoControl.SepareComponent := FALSE;
        _varInfo := __VARINFO(inoStatus.SeparatorHomePos);

        THIS^.Messenger.OnCondition(_infoTimer.Q AND NOT inoStatus.SeparatorHomePos)
            .Warning(_sb.Clear().Append('<#Waiting for #>').Append(_varInfo.Symbol).ToString());

        IF inoStatus.SeparatorHomePos THEN
            _progress := _progress + 1;
            _timer(In := FALSE);
        END_IF;
    END_IF;

    IF _progress = 2 THEN
        Messenger.Debug('<#Waiting for component in  separator#>');
        _timer(IN := inoStatus.SeparatorPresent, Pt := inoConfig.TimeToComponentInSeparator);

        IF _timer.Q THEN
            _progress := _progress + 1;
            _timer(In := FALSE);
        END_IF
    END_IF;

    IF _progress = 3 THEN
        inoControl.SepareComponent := TRUE;
        _varInfo := __VARINFO(inoStatus.SeparatorWorkPos);

        THIS^.Messenger.OnCondition(_infoTimer.Q AND NOT inoStatus.SeparatorWorkPos)
            .Warning(_sb.Clear().Append('<#Waiting for #>').Append(_varInfo.Symbol).ToString());

        IF inoStatus.SeparatorWorkPos THEN
            _progress := _progress + 1;
            _timer(In := FALSE);
        END_IF;
    END_IF;

    IF _progress = 4 THEN
        Messenger.Debug('<#Waiting for component in Pick position#>');
        _timer(IN := inoStatus.SeparatorPresent, Pt := inoConfig.TimeToComponentOutSeparator);

        IF inoStatus.SeparatorPresent THEN
            _progress := _progress + 1;
            _timer(In := FALSE);
        END_IF
    END_IF;

    IF _progress = 5 THEN
        _componentReady := TRUE;
        THIS^.DoneWhen(TRUE);
    END_IF;

    CallTimers(TRUE);
    THIS^.ThrowWhen(_errorTimer.Q);
END_IF

inoStatus.ComponentReady := _componentReady;

IF THIS^.Error AND NOT _errorMessage.Pinned THEN
    THIS^.Restore();
END_IF

PROPERTY PUBLIC ComponentReady : bool
GET
ComponentReady := _componentReady;
END_GET
END_PROPERTY

(*~
    <docu>
        <summary>
            Executes when task is aborted.
        </summary>
    </docu>
~*)
METHOD PROTECTED OnAbort
IF __ISVALIDREF(inoStatus) THEN
    THIS^.inoStatus.ActionDescription := '<#Separator task  was aborted.#>';
END_IF;
END_METHOD

(*~
    <docu>
        <summary>
            Executes when task reaches the ```Done``` state .
        </summary>
    </docu>
~*)
METHOD PROTECTED OnDone
IF __ISVALIDREF(inoStatus) THEN
    THIS^.inoStatus.ActionDescription := '<#Separator task  finished successfully.#>';
END_IF;

_progress := 0;

IF AutoRestore THEN
    Restore();
END_IF
END_METHOD

METHOD PROTECTED OnError
VAR
    description : STRING;
END_VAR
description := '<#Separator task finished with error.#>';
_componentReady := false;

IF __ISVALIDREF(inoStatus) THEN
    THIS^.inoStatus.ActionDescription := description;
END_IF;

THIS^._errorMessage.Error(_sb.Clear().Append(description).Append(' To restore acknowledge this alarm.').ToString()).Pin();
END_METHOD

METHOD PROTECTED OnStart
IF __ISVALIDREF(inoStatus) THEN
    THIS^.inoStatus.ActionDescription := '<#Separator task started.#>';
END_IF;

_componentReady := false;
CallTimers(FALSE);
END_METHOD

(*~
    <docu>
        <summary>
            Restores this instance to the Ready state. Can be called explicitly or from within one of the restore mechanisms.
            <para>
                See also <see cref="PlcDocu.TcoCore.TcoTask.AutoRestorable()"/>
            </para>
        </summary>
    </docu>
~*)
METHOD Restore : ITcoRestorable
SUPER^.Restore();
_componentReady := false;
END_METHOD

END_FUNCTION_BLOCK

// ---- POUs/Prototypes/TiconPickStep/TcoTixonPickStep_v_1_x_x.TcPOU
FUNCTION_BLOCK TcoTixonPickStep_v_1_x_x EXTENDS TcoCore.TcoComponent
VAR_INPUT
    inControllerInAuto : BOOL;
    inNotEmptyFeeder : BOOL;
    inSeparatorHomePos : BOOL;
    inFillingSensor : BOOL;
    inSeparatorPresent : BOOL;
    inStepperHomePos : BOOL;
    inStepperWorkPos : BOOL;
    inSeparatorWorkPos : BOOL;
    inPickZone : BOOL;
END_VAR
VAR_OUTPUT
    outFeedingA : BOOL;
    outSepareComponent : BOOL;
    outBlowValveA : BOOL;
    outRedLed : BOOL;
    outGreenLed : BOOL;
    outHopper : BOOL;
    outStepperValve : BOOL;
END_VAR
VAR
    {attribute addProperty Name "<#Status#>"}
    {attribute clr [ReadOnly()]}
    _status : TcoTixonPickStep_Status_v_1_x_x;
    {attribute addProperty Name "<#Control#>"}
    _control : TcoTixonPickStep_Control_v_1_x_x;
    {attribute addProperty Name "<#Config#>"}
    _config : TcoTixonPickStep_Config_v_1_x_x;
    _someTaskIsActive : BOOL;
    {attribute 'hide'}
    _blink : TcoUtilities.TcoBlinker(THIS^);
    _runAutomatic : BOOL;
    _hasError : BOOL;
END_VAR
VAR
    {attribute addProperty Name "<#Separator task#>"}
    _separatorTask : TcoTixonPickStepSeparatorTask(THIS^);
    {attribute addProperty Name "<#Buffer task#>"}
    _bufferTask : TcoTixonBufferTask(THIS^);
    {attribute addProperty Name "<#Step task#>"}
    _stepperTask : TcoTixonPickStepTask(THIS^);
    {attribute addProperty Name "<#Hopper task#>"}
    _hopperTask : TcoTixonHopperTask(THIS^);
    {attribute addProperty Name "<#Restore#>"}
    _restoreTask : TcoCore.TcoTask(THIS^);
END_VAR
VAR
    {attribute 'hide'}
    _sb : TcoCore.StringBuilder;
END_VAR

_blink(inOnTime := _config.BlinkTime, inOffTime := _config.BlinkTime);
UpdateStatus();
_separatorTask.Enabled := TRUE;
_separatorTask(inoConfig := _config, inoControl := _control, inoStatus := _status);
_bufferTask.Enabled := TRUE;
_bufferTask(inoConfig := _config, inoControl := _control, inoStatus := _status);
_stepperTask.Enabled := TRUE;
_stepperTask(inoConfig := _config, inoControl := _control, inoStatus := _status);
_hopperTask.Enabled := _config.HopperActive;
_hopperTask(inoConfig := _config, inoControl := _control, inoStatus := _status);
//*************RESTORE********************
_restoreTask.Enabled := TRUE;

IF _restoreTask.Execute() THEN
    Restore();
    _restoreTask.DoneWhen(TRUE);
END_IF
//****************************************
UpdateControl();

METHOD PUBLIC BufferFeed : TcoCore.ITcoTaskStatus
BufferFeed := _bufferTask.Invoke();
_bufferTask.AutoRestore := false;
END_METHOD

PROPERTY PUBLIC BufferTask : REFERENCE TO TcoTixonBufferTask
GET
BufferTask ref= _bufferTask;
END_GET
END_PROPERTY

(*~
    <docu>
        <summary>
            Gets the configuration of the Tixon PickStep.
        </summary>
    </docu>
~*)
PROPERTY Config : REFERENCE TO TcoTixonPickStep_Config_v_1_x_x
GET
Config REF= _config;
END_GET
END_PROPERTY

METHOD PUBLIC CyclicBufferFeed : TcoCore.ITcoTaskStatus
CyclicBufferFeed := _bufferTask.Invoke();
_bufferTask.AutoRestore := true;
END_METHOD

METHOD PUBLIC CyclicHopperFeed : TcoCore.ITcoTaskStatus
CyclicHopperFeed := _hopperTask.Invoke();
_hopperTask.AutoRestore := TRUE;
END_METHOD

METHOD PUBLIC CyclicSepare : TcoCore.ITcoTaskStatus
CyclicSepare := _separatorTask.Invoke();
_separatorTask.AutoRestore := true;
END_METHOD

METHOD PUBLIC CyclicStepperFeed : TcoCore.ITcoTaskStatus
VAR_INPUT
END_VAR
CyclicStepperFeed := _stepperTask.Invoke();
_stepperTask.AutoRestore := true;
END_METHOD

METHOD PUBLIC DefaultSignalisation
VAR_INPUT
END_VAR
// led signalisation
_hasError := _separatorTask.Error OR _stepperTask.Error OR _bufferTask.Error OR _hopperTask.Error;
_control.GreenLed := FALSE;
_control.RedLed := FALSE;

IF NOT _status.ControllerInAuto THEN
    _control.GreenLed := TRUE;
    _control.RedLed := TRUE;
ELSIF _hasError AND _blink.IsOn AND _status.ControllerInAuto THEN
    _control.RedLed := TRUE;
ELSIF _status.ControllerInAuto AND NOT _hasError AND _status.NotEmptyFeeder THEN
    _control.GreenLed := TRUE;
ELSIF _blink.IsOn AND _status.ControllerInAuto AND NOT _status.NotEmptyFeeder THEN
    _control.GreenLed := TRUE;
    _control.RedLed := TRUE;
END_IF
END_METHOD

METHOD PUBLIC HopperFeed : TcoCore.ITcoTaskStatus
HopperFeed := _hopperTask.Invoke();
_hopperTask.AutoRestore := false;
END_METHOD

PROPERTY PUBLIC HopperTask : reference TO TcoTixonHopperTask
GET
HopperTask ref= _hopperTask;
END_GET
END_PROPERTY

(*~
    <docu>
        <summary>
            Restores this instance to the Ready state. Can be called explicitly or from within one of the restore mechanisms.
        </summary>
    </docu>
~*)
METHOD Restore : ITcoRestorable
RestoreTasks();
_control.BlowAValve := FALSE;
_control.FeedingA := FALSE;
_control.GreenLed := FALSE;
_control.RedLed := FALSE;
_control.SepareComponent := FALSE;
_control.StepperValve := FALSE;
_control.Hooper := FALSE;
END_METHOD

METHOD INTERNAL RestoreTasks
//_resetTask.Restore();
_separatorTask.Restore();
_bufferTask.Restore();
_stepperTask.Restore();
_hopperTask.Restore();
END_METHOD

PROPERTY PUBLIC SeparatorTask : REFERENCE TO TcoTixonPickStepSeparatorTask
GET
SeparatorTask ref= _separatorTask;
END_GET
END_PROPERTY

METHOD PUBLIC Separe : TcoCore.ITcoTaskStatus
Separe := _separatorTask.Invoke();
_separatorTask.AutoRestore := false;
END_METHOD

(*~
    <docu>
        <summary>
            Custom service (manual, maintenance) logic.
            This method must be implemented in derived class.
        </summary>
    </docu>
~*)
METHOD PROTECTED ServiceMode
END_METHOD

(*~
    <docu>
        <summary>
            Gets the status of the Tixon PickStep.
        </summary>
    </docu>
~*)
PROPERTY Status : REFERENCE TO TcoTixonPickStep_Status_v_1_x_x
GET
Status REF= _status;
END_GET
END_PROPERTY

METHOD PUBLIC StepperFeed : TcoCore.ITcoTaskStatus
VAR_INPUT
END_VAR
StepperFeed := _stepperTask.Invoke();
_stepperTask.AutoRestore := FALSE;
END_METHOD

PROPERTY PUBLIC StepTask : REFERENCE TO TcoTixonPickStepTask
GET
StepTask ref= _stepperTask;
END_GET
END_PROPERTY

METHOD INTERNAL UpdateControl
VAR_INPUT
END_VAR
VAR
    index : INT;
END_VAR
outBlowValveA := _control.BlowAValve;
outFeedingA := _control.FeedingA;
outGreenLed := _control.GreenLed;
outRedLed := _control.RedLed;
outSepareComponent := _control.SepareComponent;
outStepperValve := _control.StepperValve;
outHopper := _control.Hooper;
END_METHOD

METHOD INTERNAL UpdateStatus
VAR
END_VAR
_status.NotEmptyFeeder := inNotEmptyFeeder;
_status.FillingSensor := inFillingSensor;
_status.SeparatorHomePos := inSeparatorHomePos;
_status.SeparatorPresent := inSeparatorPresent;
_status.SeparatorWorkPos := inSeparatorWorkPos;
_status.ControllerInAuto := inControllerInAuto;
_status.InPickZone := inPickZone;
END_METHOD

END_FUNCTION_BLOCK

// ---- POUs/Prototypes/TiconPickVibro/Taks/TcoTixonPickVibroFeederTask.TcPOU
FUNCTION_BLOCK TcoTixonPickVibroFeederTask EXTENDS TcoTixonFeedingTask
VAR_IN_OUT
    inoConfig : TcoTixonPickVibro_Config_v_1_x_x;
    inoControl : TcoTixonPickVibro_Control_v_1_x_x;
    inoStatus : TcoTixonPickVibro_Status_v_1_x_x;
END_VAR
VAR
    _timerIsFull : TON;
END_VAR

IF Execute() THEN
    _timerIsFull(IN := inoStatus.FillingSensor, PT := inoConfig.BufferFullTime);

    IF _progress = 0 THEN
        IF NOT __ISVALIDREF(inoControl) THEN
            _varInfo := __VARINFO(inoControl);
            Messenger.Programming(_sb.Clear().Append('<#Invalid reference: #>').Append(_varInfo.Symbol).ToString()).Pin();
        ELSIF NOT __ISVALIDREF(inoConfig) THEN
            _varInfo := __VARINFO(inoConfig);
            Messenger.Programming(_sb.Clear().Append('<#Invalid reference: #>').Append(_varInfo.Symbol).ToString()).Pin();
        ELSIF NOT __ISVALIDREF(inoStatus) THEN
            _varInfo := __VARINFO(inoStatus);
            Messenger.Programming(_sb.Clear().Append('<#Invalid reference: #>').Append(_varInfo.Symbol).ToString()).Pin();
        ELSIF NOT inoStatus.ControllerInAuto THEN
            _varInfo := __VARINFO(inoStatus.ControllerInAuto);
            Messenger.Warning(_sb.Clear().Append('<#Tixon control system not in auto #>').Append(_varInfo.Symbol).ToString());
        ELSE
            _progress := _progress + 1;
        END_IF
    END_IF

    IF _progress = 1 THEN
        _progress := _progress + 1;
        _timer(In := FALSE);
    END_IF;

    IF _progress = 2 THEN
        Messenger.Debug('<#Waiting for buffer empty#>');
        _timer(IN := NOT inoStatus.FillingSensor, Pt := inoConfig.BufferEmptyTime);

        IF _timer.Q AND inoControl.FeedingA THEN
            _progress := _progress + 1;
            _timer(In := FALSE);
        END_IF
    END_IF;

    IF _progress = 3 THEN
        Messenger.Debug('<#Waiting for blow B on #>');
        _timer(IN := TRUE, Pt := inoConfig.FeederBlowBStartTime);
        inoControl.BlowAValve := inoConfig.BufferBlowActive;

        IF _timer.Q THEN
            inoControl.FeedingB := inoConfig.FeederBlowBActive;
            Messenger.Debug('<#Start  vibratorating and blowing#>');
            _progress := _progress + 1;
            _timer(In := FALSE);
        END_IF;
    END_IF;

    IF _progress = 4 THEN
        Messenger.Debug('<#Waiting for buffer empty#>');

        IF _timerIsFull.Q THEN
            _progress := _progress + 1;
            _timer(In := FALSE);
        ELSE
            _progress := 3;
            _timer(In := FALSE);
        END_IF
    END_IF;

    IF _progress = 5 THEN
        inoControl.FeedingB := FALSE;
        Messenger.Debug('<#Waiting for buffer is full adn blow ending#>');
        _timer(IN := inoStatus.FillingSensor, Pt := inoConfig.FeederBlowBFullTime);

        IF _timer.Q THEN
            inoControl.BlowValveB := FALSE;
            _progress := _progress + 1;
            _timer(In := FALSE);
        END_IF;
    END_IF;

    IF _progress = 6 THEN
        THIS^.DoneWhen(TRUE);
    END_IF;

    CallTimers(TRUE);
    THIS^.ThrowWhen(_errorTimer.Q);
END_IF

IF THIS^.Error AND NOT _errorMessage.Pinned THEN
    THIS^.Restore();
END_IF

(*~
    <docu>
        <summary>
            Executes when task is aborted.
        </summary>
    </docu>
~*)
METHOD PROTECTED OnAbort
IF __ISVALIDREF(inoStatus) THEN
    THIS^.inoStatus.ActionDescription := '<#Vib. bin task  was aborted.#>';
END_IF;
END_METHOD

(*~
    <docu>
        <summary>
            Executes when task reaches the ```Done``` state .
        </summary>
    </docu>
~*)
METHOD PROTECTED OnDone
IF __ISVALIDREF(inoStatus) THEN
    THIS^.inoStatus.ActionDescription := '<#Vib. bin task  finished successfully.#>';
END_IF;

_progress := 0;

IF AutoRestore THEN
    Restore();
END_IF
END_METHOD

METHOD PROTECTED OnError
VAR
    description : STRING;
END_VAR
description := '<#Vib. bin task finished with error.#>';

IF __ISVALIDREF(inoStatus) THEN
    THIS^.inoStatus.ActionDescription := description;
END_IF;

THIS^._errorMessage.Error(_sb.Clear().Append(description).Append(' To restore acknowledge this alarm.').ToString()).Pin();
END_METHOD

METHOD PROTECTED OnStart
IF __ISVALIDREF(inoStatus) THEN
    THIS^.inoStatus.ActionDescription := '<#Vib. bin task started.#>';
END_IF;

CallTimers(FALSE);
_timerIsFull(In := FALSE);
END_METHOD

(*~
    <docu>
        <summary>
            Restores this instance to the Ready state. Can be called explicitly or from within one of the restore mechanisms.
            <para>
                See also <see cref="PlcDocu.TcoCore.TcoTask.AutoRestorable()"/>
            </para>
        </summary>
    </docu>
~*)
METHOD Restore : ITcoRestorable
SUPER^.Restore();
_timerIsFull(In := FALSE);
END_METHOD

END_FUNCTION_BLOCK

// ---- POUs/Prototypes/TiconPickVibro/Taks/TcoTixonPickVibroSeparatorTask.TcPOU
FUNCTION_BLOCK TcoTixonPickVibroSeparatorTask EXTENDS TcoTixonFeedingTask
VAR_IN_OUT
    inoConfig : TcoTixonPickVibro_Config_v_1_x_x;
    inoControl : TcoTixonPickVibro_Control_v_1_x_x;
    inoStatus : TcoTixonPickVibro_Status_v_1_x_x;
END_VAR
VAR
    _componentReady : BOOL;
END_VAR

IF Execute() THEN
    IF _progress = 0 THEN
        IF NOT __ISVALIDREF(inoControl) THEN
            _varInfo := __VARINFO(inoControl);
            Messenger.Programming(_sb.Clear().Append('<#Invalid reference: #>').Append(_varInfo.Symbol).ToString()).Pin();
        ELSIF NOT __ISVALIDREF(inoConfig) THEN
            _varInfo := __VARINFO(inoConfig);
            Messenger.Programming(_sb.Clear().Append('<#Invalid reference: #>').Append(_varInfo.Symbol).ToString()).Pin();
        ELSIF NOT __ISVALIDREF(inoStatus) THEN
            _varInfo := __VARINFO(inoStatus);
            Messenger.Programming(_sb.Clear().Append('<#Invalid reference: #>').Append(_varInfo.Symbol).ToString()).Pin();
        ELSIF NOT inoStatus.ControllerInAuto THEN
            _varInfo := __VARINFO(inoStatus.ControllerInAuto);
            Messenger.Warning(_sb.Clear().Append('<#Tixon control system not in auto #>').Append(_varInfo.Symbol).ToString());
        ELSIF NOT inoConfig.SeparatorActive THEN
            _progress := 4;
        ELSE
            _progress := _progress + 1;
        END_IF
    END_IF

    IF _progress = 1 THEN
        inoControl.SepareComponent := FALSE;
        _varInfo := __VARINFO(inoStatus.SeparatorHomePos);

        THIS^.Messenger.OnCondition(_infoTimer.Q AND NOT inoStatus.SeparatorHomePos)
            .Warning(_sb.Clear().Append('<#Waiting for #>').Append(_varInfo.Symbol).ToString());

        IF inoStatus.SeparatorHomePos THEN
            _progress := _progress + 1;
            _timer(In := FALSE);
        END_IF;
    END_IF;

    IF _progress = 2 THEN
        Messenger.Debug('<#Waiting for component in  separator#>');
        _timer(IN := inoStatus.SeparatorPresent, Pt := inoConfig.TimeToComponentInSeparator);

        IF _timer.Q THEN
            _progress := _progress + 1;
            _timer(In := FALSE);
        END_IF
    END_IF;

    IF _progress = 3 THEN
        inoControl.SepareComponent := TRUE;
        _varInfo := __VARINFO(inoStatus.SeparatorWorkPos);

        THIS^.Messenger.OnCondition(_infoTimer.Q AND NOT inoStatus.SeparatorWorkPos)
            .Warning(_sb.Clear().Append('<#Waiting for #>').Append(_varInfo.Symbol).ToString());

        IF inoStatus.SeparatorWorkPos THEN
            _progress := _progress + 1;
            _timer(In := FALSE);
        END_IF;
    END_IF;

    IF _progress = 4 THEN
        Messenger.Debug('<#Waiting for component in Pick position#>');
        _timer(IN := inoStatus.SeparatorPresent, Pt := inoConfig.TimeToComponentOutSeparator);

        IF inoStatus.SeparatorPresent THEN
            _progress := _progress + 1;
            _timer(In := FALSE);
        END_IF
    END_IF;

    IF _progress = 5 THEN
        _componentReady := TRUE;
        THIS^.DoneWhen(TRUE);
    END_IF;

    CallTimers(TRUE);
    THIS^.ThrowWhen(_errorTimer.Q);
END_IF

inoStatus.ComponentReady := _componentReady;

IF THIS^.Error AND NOT _errorMessage.Pinned THEN
    THIS^.Restore();
END_IF

PROPERTY PUBLIC ComponentReady : bool
GET
ComponentReady := _componentReady;
END_GET
END_PROPERTY

(*~
    <docu>
        <summary>
            Executes when task is aborted.
        </summary>
    </docu>
~*)
METHOD PROTECTED OnAbort
IF __ISVALIDREF(inoStatus) THEN
    THIS^.inoStatus.ActionDescription := '<#Separator task  was aborted.#>';
END_IF;
END_METHOD

(*~
    <docu>
        <summary>
            Executes when task reaches the ```Done``` state .
        </summary>
    </docu>
~*)
METHOD PROTECTED OnDone
IF __ISVALIDREF(inoStatus) THEN
    THIS^.inoStatus.ActionDescription := '<#Separator task  finished successfully.#>';
END_IF;

_progress := 0;

IF AutoRestore THEN
    Restore();
END_IF
END_METHOD

METHOD PROTECTED OnError
VAR
    description : STRING;
END_VAR
description := '<#Separator task finished with error.#>';
_componentReady := false;

IF __ISVALIDREF(inoStatus) THEN
    THIS^.inoStatus.ActionDescription := description;
END_IF;

THIS^._errorMessage.Error(_sb.Clear().Append(description).Append(' To restore acknowledge this alarm.').ToString()).Pin();
END_METHOD

METHOD PROTECTED OnStart
IF __ISVALIDREF(inoStatus) THEN
    THIS^.inoStatus.ActionDescription := '<#Separator task started.#>';
END_IF;

_componentReady := false;
CallTimers(FALSE);
END_METHOD

(*~
    <docu>
        <summary>
            Restores this instance to the Ready state. Can be called explicitly or from within one of the restore mechanisms.
            <para>
                See also <see cref="PlcDocu.TcoCore.TcoTask.AutoRestorable()"/>
            </para>
        </summary>
    </docu>
~*)
METHOD Restore : ITcoRestorable
SUPER^.Restore();
_componentReady := false;
END_METHOD

END_FUNCTION_BLOCK

// ---- POUs/Prototypes/TiconPickVibro/TcoTixonPickVibro_v_1_x_x.TcPOU
FUNCTION_BLOCK TcoTixonPickVibro_v_1_x_x EXTENDS TcoCore.TcoComponent
VAR_INPUT
    inControllerInAuto : BOOL;
    inNotEmptyFeeder : BOOL;
    inSeparatorHomePos : BOOL;
    inFillingSensor : BOOL;
    inSeparatorPresent : BOOL;
    inSeparatorWorkPos : BOOL;
    inPickZone : BOOL;
END_VAR
VAR_OUTPUT
    outFeedingA : BOOL;
    outSepareComponent : BOOL;
    outBlowValveA : BOOL;
    outRedLed : BOOL;
    outGreenLed : BOOL;
    outHopper : BOOL;
    outFeedingB : BOOL;
    outBlowValveB : BOOL;
END_VAR
VAR
    {attribute addProperty Name "<#Status#>"}
    {attribute clr [ReadOnly()]}
    _status : TcoTixonPickVibro_Status_v_1_x_x;
    {attribute addProperty Name "<#Control#>"}
    _control : TcoTixonPickVibro_Control_v_1_x_x;
    {attribute addProperty Name "<#Config#>"}
    _config : TcoTixonPickVibro_Config_v_1_x_x;
    _someTaskIsActive : BOOL;
    {attribute 'hide'}
    _blink : TcoUtilities.TcoBlinker(THIS^);
    _runAutomatic : BOOL;
    _hasError : BOOL;
END_VAR
VAR
    {attribute addProperty Name "<#Separator task#>"}
    _separatorTask : TcoTixonPickVibroSeparatorTask(THIS^);
    {attribute addProperty Name "<#Buffer task#>"}
    _bufferTask : TcoTixonBufferTask(THIS^);
    {attribute addProperty Name "<#Vibrating bin task#>"}
    _binFeederTask : TcoTixonPickVibroFeederTask(THIS^);
    {attribute addProperty Name "<#Hopper task#>"}
    _hopperTask : TcoTixonHopperTask(THIS^);
    {attribute addProperty Name "<#Restore#>"}
    _restoreTask : TcoCore.TcoTask(THIS^);
END_VAR
VAR
    {attribute 'hide'}
    _sb : TcoCore.StringBuilder;
END_VAR

_blink(inOnTime := _config.BlinkTime, inOffTime := _config.BlinkTime);
UpdateStatus();
_separatorTask.Enabled := TRUE;
_separatorTask(inoConfig := _config, inoControl := _control, inoStatus := _status);
_bufferTask.Enabled := TRUE;
_bufferTask(inoConfig := _config, inoControl := _control, inoStatus := _status);
_binFeederTask.Enabled := TRUE;
_binFeederTask(inoConfig := _config, inoControl := _control, inoStatus := _status);
_hopperTask.Enabled := _config.HopperActive;
_hopperTask(inoConfig := _config, inoControl := _control, inoStatus := _status);
//*************RESTORE********************
_restoreTask.Enabled := TRUE;

IF _restoreTask.Execute() THEN
    Restore();
    _restoreTask.DoneWhen(TRUE);
END_IF
//****************************************
UpdateControl();

METHOD PUBLIC BufferFeed : TcoCore.ITcoTaskStatus
BufferFeed := _bufferTask.Invoke();
_bufferTask.AutoRestore := false;
END_METHOD

PROPERTY PUBLIC BufferTask : REFERENCE TO TcoTixonBufferTask
GET
BufferTask ref= _bufferTask;
END_GET
END_PROPERTY

(*~
    <docu>
        <summary>
            Gets the configuration of the Tixon Step.
        </summary>
    </docu>
~*)
PROPERTY Config : REFERENCE TO TcoTixonPickVibro_Config_v_1_x_x
GET
Config REF= _config;
END_GET
END_PROPERTY

METHOD PUBLIC CyclicBinFeed : TcoCore.ITcoTaskStatus
VAR_INPUT
END_VAR
CyclicBinFeed := _binFeederTask.Invoke();
_binFeederTask.AutoRestore := true;
END_METHOD

METHOD PUBLIC CyclicBufferFeed : TcoCore.ITcoTaskStatus
CyclicBufferFeed := _bufferTask.Invoke();
_bufferTask.AutoRestore := true;
END_METHOD

METHOD PUBLIC CyclicHopperFeed : TcoCore.ITcoTaskStatus
CyclicHopperFeed := _hopperTask.Invoke();
_hopperTask.AutoRestore := TRUE;
END_METHOD

METHOD PUBLIC CyclicSepare : TcoCore.ITcoTaskStatus
CyclicSepare := _separatorTask.Invoke();
_separatorTask.AutoRestore := true;
END_METHOD

METHOD PUBLIC DefaultSignalisation
VAR_INPUT
END_VAR
// led signalisation
_hasError := _separatorTask.Error OR _bufferTask.Error OR _hopperTask.Error;
_control.GreenLed := FALSE;
_control.RedLed := FALSE;

IF NOT _status.ControllerInAuto THEN
    _control.GreenLed := TRUE;
    _control.RedLed := TRUE;
ELSIF _hasError AND _blink.IsOn AND _status.ControllerInAuto THEN
    _control.RedLed := TRUE;
ELSIF _status.ControllerInAuto AND NOT _hasError AND _status.NotEmptyFeeder THEN
    _control.GreenLed := TRUE;
ELSIF _blink.IsOn AND _status.ControllerInAuto AND NOT _status.NotEmptyFeeder THEN
    _control.GreenLed := TRUE;
    _control.RedLed := TRUE;
END_IF
END_METHOD

METHOD PUBLIC HopperFeed : TcoCore.ITcoTaskStatus
HopperFeed := _hopperTask.Invoke();
_hopperTask.AutoRestore := false;
END_METHOD

PROPERTY PUBLIC HopperTask : reference TO TcoTixonHopperTask
GET
HopperTask ref= _hopperTask;
END_GET
END_PROPERTY

(*~
    <docu>
        <summary>
            Restores this instance to the Ready state. Can be called explicitly or from within one of the restore mechanisms.
        </summary>
    </docu>
~*)
METHOD Restore : ITcoRestorable
RestoreTasks();
_control.BlowAValve := FALSE;
_control.FeedingA := FALSE;
_control.GreenLed := FALSE;
_control.RedLed := FALSE;
_control.SepareComponent := FALSE;
_control.FeedingB := FALSE;
_control.BlowValveB := FALSE;
_control.Hooper := FALSE;
END_METHOD

METHOD INTERNAL RestoreTasks
//_resetTask.Restore();
_separatorTask.Restore();
_bufferTask.Restore();
_binFeederTask.Restore();
_hopperTask.Restore();
END_METHOD

PROPERTY PUBLIC SeparatorTask : REFERENCE TO TcoTixonPickVibroSeparatorTask
GET
SeparatorTask ref= _separatorTask;
END_GET
END_PROPERTY

METHOD PUBLIC Separe : TcoCore.ITcoTaskStatus
Separe := _separatorTask.Invoke();
_separatorTask.AutoRestore := false;
END_METHOD

(*~
    <docu>
        <summary>
            Custom service (manual, maintenance) logic.
            This method must be implemented in derived class.
        </summary>
    </docu>
~*)
METHOD PROTECTED ServiceMode
END_METHOD

(*~
    <docu>
        <summary>
            Gets the status of the Tixon Step.
        </summary>
    </docu>
~*)
PROPERTY Status : REFERENCE TO TcoTixonPickVibro_Status_v_1_x_x
GET
Status REF= _status;
END_GET
END_PROPERTY

METHOD INTERNAL UpdateControl
VAR_INPUT
END_VAR
VAR
    index : INT;
END_VAR
outBlowValveA := _control.BlowAValve;
outFeedingA := _control.FeedingA;
outGreenLed := _control.GreenLed;
outRedLed := _control.RedLed;
outSepareComponent := _control.SepareComponent;
outFeedingB := _control.FeedingB;
outBlowValveB := _control.BlowValveB;
outHopper := _control.Hooper;
END_METHOD

METHOD INTERNAL UpdateStatus
VAR
END_VAR
_status.NotEmptyFeeder := inNotEmptyFeeder;
_status.FillingSensor := inFillingSensor;
_status.SeparatorHomePos := inSeparatorHomePos;
_status.SeparatorPresent := inSeparatorPresent;
_status.SeparatorWorkPos := inSeparatorWorkPos;
_status.ControllerInAuto := inControllerInAuto;
_status.InPickZone := inPickZone;
END_METHOD

END_FUNCTION_BLOCK

// ---- POUs/Prototypes/TixonPickVibroBasic/Tasks/TcoTixonPickVibroBasicSeparatorTask.TcPOU
FUNCTION_BLOCK TcoTixonPickVibroBasicSeparatorTask EXTENDS TcoTixonFeedingTask
VAR_IN_OUT
    inoConfig : TcoTixonPickVibroBasic_Config_v_1_x_x;
    inoControl : TcoTixonPickVibroBasic_Control_v_1_x_x;
    inoStatus : TcoTixonPickVibroBasic_Status_v_1_x_x;
END_VAR
VAR
    _componentReady : BOOL;
END_VAR

IF Execute() THEN
    IF _progress = 0 THEN
        IF NOT __ISVALIDREF(inoControl) THEN
            _varInfo := __VARINFO(inoControl);
            Messenger.Programming(_sb.Clear().Append('<#Invalid reference: #>').Append(_varInfo.Symbol).ToString()).Pin();
        ELSIF NOT __ISVALIDREF(inoConfig) THEN
            _varInfo := __VARINFO(inoConfig);
            Messenger.Programming(_sb.Clear().Append('<#Invalid reference: #>').Append(_varInfo.Symbol).ToString()).Pin();
        ELSIF NOT __ISVALIDREF(inoStatus) THEN
            _varInfo := __VARINFO(inoStatus);
            Messenger.Programming(_sb.Clear().Append('<#Invalid reference: #>').Append(_varInfo.Symbol).ToString()).Pin();
        ELSIF NOT inoStatus.ControllerInAuto THEN
            _varInfo := __VARINFO(inoStatus.ControllerInAuto);
            Messenger.Warning(_sb.Clear().Append('<#Tixon control system not in auto #>').Append(_varInfo.Symbol).ToString());
        ELSIF NOT inoConfig.SeparatorActive THEN
            _progress := 4;
        ELSE
            _progress := _progress + 1;
        END_IF
    END_IF

    IF _progress = 1 THEN
        inoControl.SepareComponent := FALSE;
        _varInfo := __VARINFO(inoStatus.SeparatorHomePos);

        THIS^.Messenger.OnCondition(_infoTimer.Q AND NOT inoStatus.SeparatorHomePos)
            .Warning(_sb.Clear().Append('<#Waiting for #>').Append(_varInfo.Symbol).ToString());

        IF inoStatus.SeparatorHomePos THEN
            _progress := _progress + 1;
            _timer(In := FALSE);
        END_IF;
    END_IF;

    IF _progress = 2 THEN
        Messenger.Debug('<#Waiting for component in  separator#>');
        _timer(IN := inoStatus.SeparatorPresent, Pt := inoConfig.TimeToComponentInSeparator);

        IF _timer.Q THEN
            _progress := _progress + 1;
            _timer(In := FALSE);
        END_IF
    END_IF;

    IF _progress = 3 THEN
        inoControl.SepareComponent := TRUE;
        _varInfo := __VARINFO(inoStatus.SeparatorWorkPos);

        THIS^.Messenger.OnCondition(_infoTimer.Q AND NOT inoStatus.SeparatorWorkPos)
            .Warning(_sb.Clear().Append('<#Waiting for #>').Append(_varInfo.Symbol).ToString());

        IF inoStatus.SeparatorWorkPos THEN
            _progress := _progress + 1;
            _timer(In := FALSE);
        END_IF;
    END_IF;

    IF _progress = 4 THEN
        Messenger.Debug('<#Waiting for component in Pick position#>');
        _timer(IN := inoStatus.SeparatorPresent, Pt := inoConfig.TimeToComponentOutSeparator);

        IF inoStatus.SeparatorPresent THEN
            _progress := _progress + 1;
            _timer(In := FALSE);
        END_IF
    END_IF;

    IF _progress = 5 THEN
        _componentReady := TRUE;
        THIS^.DoneWhen(TRUE);
    END_IF;

    CallTimers(TRUE);
    THIS^.ThrowWhen(_errorTimer.Q);
END_IF

inoStatus.ComponentReady := _componentReady;

IF THIS^.Error AND NOT _errorMessage.Pinned THEN
    THIS^.Restore();
END_IF

PROPERTY PUBLIC ComponentReady : bool
GET
ComponentReady := _componentReady;
END_GET
END_PROPERTY

(*~
    <docu>
        <summary>
            Executes when task is aborted.
        </summary>
    </docu>
~*)
METHOD PROTECTED OnAbort
IF __ISVALIDREF(inoStatus) THEN
    THIS^.inoStatus.ActionDescription := '<#Separator task  was aborted.#>';
END_IF;
END_METHOD

(*~
    <docu>
        <summary>
            Executes when task reaches the ```Done``` state .
        </summary>
    </docu>
~*)
METHOD PROTECTED OnDone
IF __ISVALIDREF(inoStatus) THEN
    THIS^.inoStatus.ActionDescription := '<#Separator task  finished successfully.#>';
END_IF;

_progress := 0;

IF AutoRestore THEN
    Restore();
END_IF
END_METHOD

METHOD PROTECTED OnError
VAR
    description : STRING;
END_VAR
description := '<#Separator task finished with error.#>';
_componentReady := false;

IF __ISVALIDREF(inoStatus) THEN
    THIS^.inoStatus.ActionDescription := description;
END_IF;

THIS^._errorMessage.Error(_sb.Clear().Append(description).Append(' To restore acknowledge this alarm.').ToString()).Pin();
END_METHOD

METHOD PROTECTED OnStart
IF __ISVALIDREF(inoStatus) THEN
    THIS^.inoStatus.ActionDescription := '<#Separator task started.#>';
END_IF;

_componentReady := false;
CallTimers(FALSE);
END_METHOD

(*~
    <docu>
        <summary>
            Restores this instance to the Ready state. Can be called explicitly or from within one of the restore mechanisms.
            <para>
                See also <see cref="PlcDocu.TcoCore.TcoTask.AutoRestorable()"/>
            </para>
        </summary>
    </docu>
~*)
METHOD Restore : ITcoRestorable
SUPER^.Restore();
_componentReady := false;
END_METHOD

END_FUNCTION_BLOCK

// ---- POUs/Prototypes/TixonPickVibroBasic/TcoTixonPickVibroBasic_v_1_x_x.TcPOU
FUNCTION_BLOCK TcoTixonPickVibroBasic_v_1_x_x EXTENDS TcoCore.TcoComponent
VAR_INPUT
    inControllerInAuto : BOOL;
    inNotEmptyFeeder : BOOL;
    inSeparatorHomePos : BOOL;
    inFillingSensor : BOOL;
    inSeparatorPresent : BOOL;
    inSeparatorWorkPos : BOOL;
    inPickZone : BOOL;
END_VAR
VAR_OUTPUT
    outFeedingA : BOOL;
    outSepareComponent : BOOL;
    outBlowValveA : BOOL;
    outRedLed : BOOL;
    outGreenLed : BOOL;
    outHopper : BOOL;
END_VAR
VAR
    {attribute addProperty Name "<#Status#>"}
    {attribute clr [ReadOnly()]}
    _status : TcoTixonPickVibroBasic_Status_v_1_x_x;
    {attribute addProperty Name "<#Control#>"}
    _control : TcoTixonPickVibroBasic_Control_v_1_x_x;
    {attribute addProperty Name "<#Config#>"}
    _config : TcoTixonPickVibroBasic_Config_v_1_x_x;
    _someTaskIsActive : BOOL;
    {attribute 'hide'}
    _blink : TcoUtilities.TcoBlinker(THIS^);
    _runAutomatic : BOOL;
    _hasError : BOOL;
END_VAR
VAR
    {attribute addProperty Name "<#Separator task#>"}
    _separatorTask : TcoTixonPickVibroBasicSeparatorTask(THIS^);
    {attribute addProperty Name "<#Buffer task#>"}
    _bufferTask : TcoTixonBufferTask(THIS^);
    {attribute addProperty Name "<#Hopper task#>"}
    _hopperTask : TcoTixonHopperTask(THIS^);
    {attribute addProperty Name "<#Restore#>"}
    _restoreTask : TcoCore.TcoTask(THIS^);
END_VAR
VAR
    {attribute 'hide'}
    _sb : TcoCore.StringBuilder;
END_VAR

_blink(inOnTime := _config.BlinkTime, inOffTime := _config.BlinkTime);
UpdateStatus();
_separatorTask.Enabled := TRUE;
_separatorTask(inoConfig := _config, inoControl := _control, inoStatus := _status);
_bufferTask.Enabled := TRUE;
_bufferTask(inoConfig := _config, inoControl := _control, inoStatus := _status);
_hopperTask.Enabled := _config.HopperActive;
_hopperTask(inoConfig := _config, inoControl := _control, inoStatus := _status);
//*************RESTORE********************
_restoreTask.Enabled := TRUE;

IF _restoreTask.Execute() THEN
    Restore();
    _restoreTask.DoneWhen(TRUE);
END_IF
//****************************************
UpdateControl();

METHOD PUBLIC BufferFeed : TcoCore.ITcoTaskStatus
BufferFeed := _bufferTask.Invoke();
_bufferTask.AutoRestore := false;
END_METHOD

PROPERTY PUBLIC BufferTask : REFERENCE TO TcoTixonBufferTask
GET
BufferTask ref= _bufferTask;
END_GET
END_PROPERTY

(*~
    <docu>
        <summary>
            Gets the configuration of the Tixon Step.
        </summary>
    </docu>
~*)
PROPERTY Config : REFERENCE TO TcoTixonPickVibroBasic_Config_v_1_x_x
GET
Config REF= _config;
END_GET
END_PROPERTY

METHOD PUBLIC CyclicBufferFeed : TcoCore.ITcoTaskStatus
CyclicBufferFeed := _bufferTask.Invoke();
_bufferTask.AutoRestore := true;
END_METHOD

METHOD PUBLIC CyclicHopperFeed : TcoCore.ITcoTaskStatus
CyclicHopperFeed := _hopperTask.Invoke();
_hopperTask.AutoRestore := TRUE;
END_METHOD

METHOD PUBLIC CyclicSepare : TcoCore.ITcoTaskStatus
CyclicSepare := _separatorTask.Invoke();
_separatorTask.AutoRestore := true;
END_METHOD

METHOD PUBLIC DefaultSignalisation
VAR_INPUT
END_VAR
// led signalisation
_hasError := _separatorTask.Error OR _bufferTask.Error OR _hopperTask.Error;
_control.GreenLed := FALSE;
_control.RedLed := FALSE;

IF NOT _status.ControllerInAuto THEN
    _control.GreenLed := TRUE;
    _control.RedLed := TRUE;
ELSIF _hasError AND _blink.IsOn AND _status.ControllerInAuto THEN
    _control.RedLed := TRUE;
ELSIF _status.ControllerInAuto AND NOT _hasError AND _status.NotEmptyFeeder THEN
    _control.GreenLed := TRUE;
ELSIF _blink.IsOn AND _status.ControllerInAuto AND NOT _status.NotEmptyFeeder THEN
    _control.GreenLed := TRUE;
    _control.RedLed := TRUE;
END_IF
END_METHOD

METHOD PUBLIC HopperFeed : TcoCore.ITcoTaskStatus
HopperFeed := _hopperTask.Invoke();
_hopperTask.AutoRestore := false;
END_METHOD

PROPERTY PUBLIC HopperTask : reference TO TcoTixonHopperTask
GET
HopperTask ref= _hopperTask;
END_GET
END_PROPERTY

(*~
    <docu>
        <summary>
            Restores this instance to the Ready state. Can be called explicitly or from within one of the restore mechanisms.
        </summary>
    </docu>
~*)
METHOD Restore : ITcoRestorable
RestoreTasks();
_control.BlowAValve := FALSE;
_control.FeedingA := FALSE;
_control.GreenLed := FALSE;
_control.RedLed := FALSE;
_control.SepareComponent := FALSE;
_control.Hooper := FALSE;
END_METHOD

METHOD INTERNAL RestoreTasks
//_resetTask.Restore();
_separatorTask.Restore();
_bufferTask.Restore();
_hopperTask.Restore();
END_METHOD

PROPERTY PUBLIC SeparatorTask : REFERENCE TO TcoTixonPickVibroBasicSeparatorTask
GET
SeparatorTask ref= _separatorTask;
END_GET
END_PROPERTY

METHOD PUBLIC Separe : TcoCore.ITcoTaskStatus
Separe := _separatorTask.Invoke();
_separatorTask.AutoRestore := false;
END_METHOD

(*~
    <docu>
        <summary>
            Custom service (manual, maintenance) logic.
            This method must be implemented in derived class.
        </summary>
    </docu>
~*)
METHOD PROTECTED ServiceMode
END_METHOD

(*~
    <docu>
        <summary>
            Gets the status of the Tixon Step.
        </summary>
    </docu>
~*)
PROPERTY Status : REFERENCE TO TcoTixonPickVibroBasic_Status_v_1_x_x
GET
Status REF= _status;
END_GET
END_PROPERTY

METHOD INTERNAL UpdateControl
VAR_INPUT
END_VAR
VAR
    index : INT;
END_VAR
outBlowValveA := _control.BlowAValve;
outFeedingA := _control.FeedingA;
outGreenLed := _control.GreenLed;
outRedLed := _control.RedLed;
outSepareComponent := _control.SepareComponent;
outHopper := _control.Hooper;
END_METHOD

METHOD INTERNAL UpdateStatus
VAR
END_VAR
_status.NotEmptyFeeder := inNotEmptyFeeder;
_status.SeparatorHomePos := inSeparatorHomePos;
_status.SeparatorPresent := inSeparatorPresent;
_status.FillingSensor := inFillingSensor;
_status.SeparatorWorkPos := inSeparatorWorkPos;
_status.ControllerInAuto := inControllerInAuto;
_status.InPickZone := inPickZone;
END_METHOD

END_FUNCTION_BLOCK

// ---- POUs/Prototypes/TixonStep/Tasks/Separe/TcoTixonStepSeparatorTask.TcPOU
FUNCTION_BLOCK TcoTixonStepSeparatorTask EXTENDS TcoTixonFeedingTask
VAR_IN_OUT
    inoConfig : TcoTixonStep_Config_v_1_x_x;
    inoControl : TcoTixonStep_Control_v_1_x_x;
    inoStatus : TcoTixonStep_Status_v_1_x_x;
END_VAR
VAR
    _componentReady : BOOL;
END_VAR

IF Execute() THEN
    IF _progress = 0 THEN
        IF NOT __ISVALIDREF(inoControl) THEN
            _varInfo := __VARINFO(inoControl);
            Messenger.Programming(_sb.Clear().Append('<#Invalid reference: #>').Append(_varInfo.Symbol).ToString()).Pin();
        ELSIF NOT __ISVALIDREF(inoConfig) THEN
            _varInfo := __VARINFO(inoConfig);
            Messenger.Programming(_sb.Clear().Append('<#Invalid reference: #>').Append(_varInfo.Symbol).ToString()).Pin();
        ELSIF NOT __ISVALIDREF(inoStatus) THEN
            _varInfo := __VARINFO(inoStatus);
            Messenger.Programming(_sb.Clear().Append('<#Invalid reference: #>').Append(_varInfo.Symbol).ToString()).Pin();
        ELSIF NOT inoStatus.ControllerInAuto THEN
            _varInfo := __VARINFO(inoStatus.ControllerInAuto);
            Messenger.Warning(_sb.Clear().Append('<#Tixon control system not in auto #>').Append(_varInfo.Symbol).ToString());
        ELSE
            IF NOT inoConfig.OutOfBoxSensorDisabled AND inoConfig.SeparatorHasWorkPosition THEN
                Messenger.Error(_sb.Clear()
                        .Append('<#Tixon has inconsistent configuration! (OutOfBoxSensorDisabled is not disabled instead of SeparatorHasWorkPosition is On!)#>')
                        .ToString()).Pin();
            ELSE
                IF NOT THIS^._errorMessage.Pinned THEN
                    _progress := _progress + 1;
                END_IF;
            END_IF;
        END_IF
    END_IF

    IF _progress = 1 THEN
        inoControl.SepareComponent := FALSE;
        _varInfo := __VARINFO(inoStatus.SeparatorHomePos);

        THIS^.Messenger.OnCondition(_infoTimer.Q AND NOT inoStatus.SeparatorHomePos)
            .Warning(_sb.Clear().Append('<#Waiting for #>').Append(_varInfo.Symbol).ToString());

        THIS^.Messenger.OnCondition(_infoTimer.Q AND inoStatus.ComponentOutOfBox AND NOT inoConfig.OutOfBoxSensorDisabled)
            .Error(_sb.Clear()
                .Append('<#Check component at the separator output. The component is probably stuck!.#>')
                .Append(_varInfo.Symbol)
                .ToString()).Pin();

        IF _infoTimer.Q AND inoStatus.ComponentOutOfBox and NOT inoConfig.OutOfBoxSensorDisabled THEN
            THIS^.ThrowWhen(_errorTimer.Q);
        ELSIF inoStatus.SeparatorHomePos AND NOT inoStatus.ComponentOutOfBox THEN
            _progress := _progress + 1;
            _timer(In := FALSE);
        END_IF;
    END_IF;

    IF _progress = 2 THEN
        Messenger.Debug('<#Waiting for component in  separator#>');
        _timer(IN := inoStatus.SeparatorPresent, Pt := inoConfig.TimeToComponentInSeparator);

        IF _timer.Q THEN
            _progress := _progress + 1;
            _timer(In := FALSE);
        END_IF
    END_IF;

    IF _progress = 3 THEN
        inoControl.SepareComponent := TRUE;
        Messenger.OnCondition(NOT inoConfig.OutOfBoxSensorDisabled).Debug('<#Waiting for component out of  separator#>');

        Messenger.OnCondition(inoConfig.OutOfBoxSensorDisabled AND inoConfig.SeparatorHasWorkPosition)
            .Warning('<#Waiting to separator to reach work position.#>');

        _timer(IN := inoStatus.SeparatorPresent, Pt := inoConfig.TimeToComponentOutSeparator);

        IF inoStatus.ComponentOutOfBox AND NOT inoConfig.OutOfBoxSensorDisabled THEN
            _progress := _progress + 1;
            _timer(In := FALSE);
        ELSIF inoConfig.OutOfBoxSensorDisabled AND inoConfig.SeparatorHasWorkPosition AND inoStatus.SeparatorWorkPos THEN
            _progress := _progress + 1;
            _timer(In := FALSE);
        ELSIF inoConfig.OutOfBoxSensorDisabled AND NOT inoConfig.SeparatorHasWorkPosition AND _timer.Q THEN
            _progress := _progress + 1;
            _timer(In := FALSE);
        ELSIF _timer.Q AND NOT inoConfig.OutOfBoxSensorDisabled THEN
            _progress := 1;
            _timer(In := FALSE);
        END_IF
    END_IF;

    IF _progress = 4 THEN
        _componentReady := TRUE;
        THIS^.DoneWhen(TRUE);
    END_IF;

    CallTimers(TRUE);
    THIS^.ThrowWhen(_errorTimer.Q);
END_IF

inoStatus.ComponentReady := _componentReady;

IF THIS^.Error AND NOT _errorMessage.Pinned THEN
    THIS^.Restore();
END_IF

PROPERTY PUBLIC ComponentReady : bool
GET
ComponentReady := _componentReady;
END_GET
END_PROPERTY

(*~
    <docu>
        <summary>
            Executes when task is aborted.
        </summary>
    </docu>
~*)
METHOD PROTECTED OnAbort
IF __ISVALIDREF(inoStatus) THEN
    THIS^.inoStatus.ActionDescription := '<#Separator task  was aborted.#>';
END_IF;
END_METHOD

(*~
    <docu>
        <summary>
            Executes when task reaches the ```Done``` state .
        </summary>
    </docu>
~*)
METHOD PROTECTED OnDone
IF __ISVALIDREF(inoStatus) THEN
    THIS^.inoStatus.ActionDescription := '<#Separator task  finished successfully.#>';
END_IF;

_progress := 0;

IF AutoRestore THEN
    Restore();
END_IF
END_METHOD

METHOD PROTECTED OnError
VAR
    description : STRING;
END_VAR
description := '<#Separator task finished with error.#>';
_componentReady := FALSE;
inoControl.SepareComponent := false;

IF __ISVALIDREF(inoStatus) THEN
    THIS^.inoStatus.ActionDescription := description;
END_IF;

THIS^._errorMessage.Error(_sb.Clear().Append(description).Append(' To restore acknowledge this alarm.').ToString()).Pin();
END_METHOD

METHOD PROTECTED OnStart
IF __ISVALIDREF(inoStatus) THEN
    THIS^.inoStatus.ActionDescription := '<#Separator task started.#>';
END_IF;

_componentReady := false;
CallTimers(FALSE);
END_METHOD

(*~
    <docu>
        <summary>
            Restores this instance to the Ready state. Can be called explicitly or from within one of the restore mechanisms.
            <para>
                See also <see cref="PlcDocu.TcoCore.TcoTask.AutoRestorable()"/>
            </para>
        </summary>
    </docu>
~*)
METHOD Restore : ITcoRestorable
SUPER^.Restore();
_componentReady := false;
END_METHOD

END_FUNCTION_BLOCK

// ---- POUs/Prototypes/TixonStep/Tasks/Step/TcoTixonStepTask.TcPOU
FUNCTION_BLOCK TcoTixonStepTask EXTENDS TcoTixonFeedingTask
VAR_IN_OUT
    inoConfig : TcoTixonStep_Config_v_1_x_x;
    inoControl : TcoTixonStep_Control_v_1_x_x;
    inoStatus : TcoTixonStep_Status_v_1_x_x;
END_VAR
VAR
    _timerIsFull : TON;
    _timerIsStucked : TON;
END_VAR

IF Execute() THEN
    _timerIsFull(IN := inoStatus.FillingSensor, PT := inoConfig.BufferFullTime);

    IF _progress = 0 THEN
        IF NOT __ISVALIDREF(inoControl) THEN
            _varInfo := __VARINFO(inoControl);
            Messenger.Programming(_sb.Clear().Append('<#Invalid reference: #>').Append(_varInfo.Symbol).ToString()).Pin();
        ELSIF NOT __ISVALIDREF(inoConfig) THEN
            _varInfo := __VARINFO(inoConfig);
            Messenger.Programming(_sb.Clear().Append('<#Invalid reference: #>').Append(_varInfo.Symbol).ToString()).Pin();
        ELSIF NOT __ISVALIDREF(inoStatus) THEN
            _varInfo := __VARINFO(inoStatus);
            Messenger.Programming(_sb.Clear().Append('<#Invalid reference: #>').Append(_varInfo.Symbol).ToString()).Pin();
        ELSIF NOT inoStatus.ControllerInAuto THEN
            _varInfo := __VARINFO(inoStatus.ControllerInAuto);
            Messenger.Warning(_sb.Clear().Append('<#Tixon control system not in auto #>').Append(_varInfo.Symbol).ToString());
        ELSE
            IF NOT THIS^._errorMessage.Pinned THEN
                _progress := _progress + 1;
            END_IF;
        END_IF
    END_IF

    IF _progress = 1 THEN
        Messenger.Debug('<#Waiting for buffer empty#>');
        _timer(IN := NOT inoStatus.FillingSensor, Pt := inoConfig.BufferEmptyTime);

        _timerIsStucked(in := inoConfig.BufferStuckedOnFillingSensor <> T#0S AND
                inoControl.FeedingA AND
                inoStatus.FillingSensor AND
                NOT inoStatus.SeparatorPresent,
            Pt := inoConfig.BufferStuckedOnFillingSensor);

        IF _timer.Q AND inoControl.FeedingA THEN
            _progress := _progress + 1;
            _timer(In := FALSE);
        ELSIF _timerIsStucked.Q AND inoControl.FeedingA AND inoStatus.FillingSensor AND NOT inoStatus.SeparatorPresent THEN
            _progress := _progress + 1;
            _timer(In := FALSE);
        END_IF
    END_IF;

    IF _progress = 2 THEN
        inoControl.StepperValve := FALSE;
        Messenger.Debug('<#Stepper to home#>');
        _timer(IN := inoStatus.StepperHomePos, Pt := inoConfig.SteperInHomeTime);

        IF _timer.Q THEN
            _progress := _progress + 1;
            _timer(In := FALSE);
        END_IF
    END_IF;

    IF _progress = 3 THEN
        inoControl.StepperValve := TRUE;
        Messenger.Debug('<#Stepper to work#>');
        _timer(IN := inoStatus.StepperWorkPos, Pt := inoConfig.SteperInWorkTime);

        IF _timer.Q THEN
            _progress := _progress + 1;
            _timer(In := FALSE);
        END_IF
    END_IF;

    IF _progress = 4 THEN
        Messenger.Debug('<#Waiting for buffer full#>');

        IF _timerIsFull.Q THEN
            _progress := _progress + 1;
            _timer(In := FALSE);
        ELSE
            _progress := 2;
            _timer(In := FALSE);
        END_IF
    END_IF;

    IF _progress = 5 THEN
        THIS^.DoneWhen(TRUE);
    END_IF;

    CallTimers(_progress > 1); //empty and strat feeding
    THIS^.ThrowWhen(_errorTimer.Q);
END_IF

IF THIS^.Error AND NOT _errorMessage.Pinned THEN
    THIS^.Restore();
END_IF

(*~
    <docu>
        <summary>
            Executes when task is aborted.
        </summary>
    </docu>
~*)
METHOD PROTECTED OnAbort
IF __ISVALIDREF(inoStatus) THEN
    THIS^.inoStatus.ActionDescription := '<#Stepper task  was aborted.#>';
END_IF;
END_METHOD

(*~
    <docu>
        <summary>
            Executes when task reaches the ```Done``` state .
        </summary>
    </docu>
~*)
METHOD PROTECTED OnDone
IF __ISVALIDREF(inoStatus) THEN
    THIS^.inoStatus.ActionDescription := '<#Stepper task  finished successfully.#>';
END_IF;

_progress := 0;

IF AutoRestore THEN
    Restore();
END_IF
END_METHOD

METHOD PROTECTED OnError
VAR
    description : STRING;
END_VAR
description := '<#Stepper task finished with error.#>';
inoControl.StepperValve := false;

IF __ISVALIDREF(inoStatus) THEN
    THIS^.inoStatus.ActionDescription := description;
END_IF;

THIS^._errorMessage.Error(_sb.Clear().Append(description).Append(' To restore acknowledge this alarm.').ToString()).Pin();
END_METHOD

METHOD PROTECTED OnStart
IF __ISVALIDREF(inoStatus) THEN
    THIS^.inoStatus.ActionDescription := '<#Stepper task started.#>';
END_IF;

CallTimers(FALSE);
_timerIsFull(In := FALSE);
_timerIsStucked(in := FALSE);
END_METHOD

(*~
    <docu>
        <summary>
            Restores this instance to the Ready state. Can be called explicitly or from within one of the restore mechanisms.
            <para>
                See also <see cref="PlcDocu.TcoCore.TcoTask.AutoRestorable()"/>
            </para>
        </summary>
    </docu>
~*)
METHOD Restore : ITcoRestorable
SUPER^.Restore();
_timerIsFull(In := FALSE);
_timerIsStucked(in := FALSE);
END_METHOD

END_FUNCTION_BLOCK

// ---- POUs/Prototypes/TixonStep/TcoTixonStep_v_1_x_x.TcPOU
FUNCTION_BLOCK TcoTixonStep_v_1_x_x EXTENDS TcoCore.TcoComponent
VAR_INPUT
    inControllerInAuto : BOOL;
    inNotEmptyFeeder : BOOL;
    inSeparatorHomePos : BOOL;
    inFillingSensor : BOOL;
    inSeparatorPresent : BOOL;
    inStepperHomePos : BOOL;
    inStepperWorkPos : BOOL;
    inComponentOutOfBox : BOOL;
    inSeparatorWorkPos : BOOL;
END_VAR
VAR_OUTPUT
    outFeedingA : BOOL;
    outSepareComponent : BOOL;
    outBlowValveA : BOOL;
    outRedLed : BOOL;
    outGreenLed : BOOL;
    outHopper : BOOL;
    outShotComponent : BOOL;
    outStepperValve : BOOL;
END_VAR
VAR
    {attribute addProperty Name "<#Status#>"}
    {attribute clr [ReadOnly()]}
    _status : TcoTixonStep_Status_v_1_x_x;
    {attribute addProperty Name "<#Control#>"}
    _control : TcoTixonStep_Control_v_1_x_x;
    {attribute addProperty Name "<#Config#>"}
    _config : TcoTixonStep_Config_v_1_x_x;
    _someTaskIsActive : BOOL;
    {attribute 'hide'}
    _blink : TcoUtilities.TcoBlinker(THIS^);
    _runAutomatic : BOOL;
    _hasError : BOOL;
END_VAR
VAR
    {attribute addProperty Name "<#Separator task#>"}
    _separatorTask : TcoTixonStepSeparatorTask(THIS^);
    {attribute addProperty Name "<#Buffer task#>"}
    _bufferTask : TcoTixonBufferTask(THIS^);
    {attribute addProperty Name "<#Step task#>"}
    _stepperTask : TcoTixonStepTask(THIS^);
    {attribute addProperty Name "<#Hopper task#>"}
    _hopperTask : TcoTixonHopperTask(THIS^);
    {attribute addProperty Name "<#Restore#>"}
    _restoreTask : TcoCore.TcoTask(THIS^);
END_VAR
VAR
    {attribute 'hide'}
    _sb : TcoCore.StringBuilder;
END_VAR

_blink(inOnTime := _config.BlinkTime, inOffTime := _config.BlinkTime);
UpdateStatus();
_separatorTask.Enabled := TRUE;
_separatorTask.ErrorTime := _config.ErrorTimeSeparator;
_separatorTask(inoConfig := _config, inoControl := _control, inoStatus := _status);
_bufferTask.Enabled := TRUE;
_bufferTask.ErrorTime := _config.ErrorTimeBuffer;
_bufferTask(inoConfig := _config, inoControl := _control, inoStatus := _status);
_stepperTask.Enabled := TRUE;
_stepperTask.ErrorTime := _config.ErrorTimeStepper;
_stepperTask(inoConfig := _config, inoControl := _control, inoStatus := _status);
_hopperTask.ErrorTime := _config.ErrorTimeHopper;
_hopperTask.Enabled := _config.HopperActive;
_hopperTask(inoConfig := _config, inoControl := _control, inoStatus := _status);
//*************RESTORE********************
_restoreTask.Enabled := TRUE;

IF _restoreTask.Execute() THEN
    Restore();
    _restoreTask.DoneWhen(TRUE);
END_IF
//****************************************
UpdateControl();

METHOD PUBLIC BufferFeed : TcoCore.ITcoTaskStatus
BufferFeed := _bufferTask.Invoke();
_bufferTask.AutoRestore := false;
END_METHOD

PROPERTY PUBLIC BufferTask : REFERENCE TO TcoTixonBufferTask
GET
BufferTask ref= _bufferTask;
END_GET
END_PROPERTY

(*~
    <docu>
        <summary>
            Gets the configuration of the Tixon Step.
        </summary>
    </docu>
~*)
PROPERTY Config : REFERENCE TO TcoTixonStep_Config_v_1_x_x
GET
Config REF= _config;
END_GET
END_PROPERTY

METHOD PUBLIC CyclicBufferFeed : TcoCore.ITcoTaskStatus
CyclicBufferFeed := _bufferTask.Invoke();
_bufferTask.AutoRestore := true;
END_METHOD

METHOD PUBLIC CyclicHopperFeed : TcoCore.ITcoTaskStatus
CyclicHopperFeed := _hopperTask.Invoke();
_hopperTask.AutoRestore := TRUE;
END_METHOD

METHOD PUBLIC CyclicSepare : TcoCore.ITcoTaskStatus
CyclicSepare := _separatorTask.Invoke();
_separatorTask.AutoRestore := true;
END_METHOD

METHOD PUBLIC CyclicStepperFeed : TcoCore.ITcoTaskStatus
VAR_INPUT
END_VAR
CyclicStepperFeed := _stepperTask.Invoke();
_stepperTask.AutoRestore := true;
END_METHOD

METHOD PUBLIC DefaultSignalisation
VAR_INPUT
END_VAR
// led signalisation
_hasError := _separatorTask.Error OR _stepperTask.Error OR _bufferTask.Error OR _hopperTask.Error;
_control.GreenLed := FALSE;
_control.RedLed := FALSE;

IF NOT _status.ControllerInAuto THEN
    _control.GreenLed := TRUE;
    _control.RedLed := TRUE;
ELSIF _hasError AND _blink.IsOn AND _status.ControllerInAuto THEN
    _control.RedLed := TRUE;
ELSIF _status.ControllerInAuto AND NOT _hasError AND _status.NotEmptyFeeder THEN
    _control.GreenLed := TRUE;
ELSIF _blink.IsOn AND _status.ControllerInAuto AND NOT _status.NotEmptyFeeder THEN
    _control.GreenLed := TRUE;
    _control.RedLed := TRUE;
END_IF
END_METHOD

METHOD PUBLIC HopperFeed : TcoCore.ITcoTaskStatus
HopperFeed := _hopperTask.Invoke();
_hopperTask.AutoRestore := false;
END_METHOD

PROPERTY PUBLIC HopperTask : reference TO TcoTixonHopperTask
GET
HopperTask ref= _hopperTask;
END_GET
END_PROPERTY

METHOD PUBLIC Push
VAR_INPUT
    inReqOn : BOOL;
END_VAR
_control.ShotComponent := inReqOn;
END_METHOD

(*~
    <docu>
        <summary>
            Restores this instance to the Ready state. Can be called explicitly or from within one of the restore mechanisms.
        </summary>
    </docu>
~*)
METHOD Restore : ITcoRestorable
RestoreTasks();
_control.BlowAValve := FALSE;
_control.FeedingA := FALSE;
_control.GreenLed := FALSE;
_control.RedLed := FALSE;
_control.SepareComponent := FALSE;
_control.StepperValve := FALSE;
_control.ShotComponent := FALSE;
_control.Hooper := FALSE;
END_METHOD

METHOD INTERNAL RestoreTasks
_separatorTask.Restore();
_bufferTask.Restore();
_stepperTask.Restore();
_hopperTask.Restore();
END_METHOD

PROPERTY PUBLIC SeparatorTask : REFERENCE TO TcoTixonStepSeparatorTask
GET
SeparatorTask ref= _separatorTask;
END_GET
END_PROPERTY

METHOD PUBLIC Separe : TcoCore.ITcoTaskStatus
Separe := _separatorTask.Invoke();
_separatorTask.AutoRestore := false;
END_METHOD

(*~
    <docu>
        <summary>
            Custom service (manual, maintenance) logic.
            This method must be implemented in derived class.
        </summary>
    </docu>
~*)
METHOD PROTECTED ServiceMode
END_METHOD

(*~
    <docu>
        <summary>
            Gets the status of the Tixon Step.
        </summary>
    </docu>
~*)
PROPERTY Status : REFERENCE TO TcoTixonStep_Status_v_1_x_x
GET
Status REF= _status;
END_GET
END_PROPERTY

METHOD PUBLIC StepperFeed : TcoCore.ITcoTaskStatus
VAR_INPUT
END_VAR
StepperFeed := _stepperTask.Invoke();
_stepperTask.AutoRestore := FALSE;
END_METHOD

PROPERTY PUBLIC StepTask : REFERENCE TO TcoTixonStepTask
GET
StepTask ref= _stepperTask;
END_GET
END_PROPERTY

METHOD INTERNAL UpdateControl
VAR_INPUT
END_VAR
VAR
    index : INT;
END_VAR
outBlowValveA := _control.BlowAValve;
outFeedingA := _control.FeedingA;
outGreenLed := _control.GreenLed;
outRedLed := _control.RedLed;
outSepareComponent := _control.SepareComponent;
outStepperValve := _control.StepperValve;
outShotComponent := _control.ShotComponent;
outHopper := _control.Hooper;
END_METHOD

METHOD INTERNAL UpdateStatus
VAR
END_VAR
_status.ComponentOutOfBox := inComponentOutOfBox;
_status.NotEmptyFeeder := inNotEmptyFeeder;
_status.FillingSensor := inFillingSensor;
_status.SeparatorHomePos := inSeparatorHomePos;
_status.SeparatorPresent := inSeparatorPresent;
_status.StepperHomePos := inStepperHomePos;
_status.StepperWorkPos := inStepperWorkPos;
_status.ControllerInAuto := inControllerInAuto;
_status.SeparatorWorkPos := inSeparatorWorkPos;
END_METHOD

END_FUNCTION_BLOCK

// ---- POUs/Prototypes/TixonVibro/Tasks/Separe/TcoTixonVibroSeparatorTask.TcPOU
FUNCTION_BLOCK TcoTixonVibroSeparatorTask EXTENDS TcoTixonFeedingTask
VAR_IN_OUT
    inoConfig : TcoTixonVibro_Config_v_1_x_x;
    inoControl : TcoTixonVibro_Control_v_1_x_x;
    inoStatus : TcoTixonVibro_Status_v_1_x_x;
END_VAR
VAR
    _componentReady : BOOL;
END_VAR

IF Execute() THEN
    IF _progress = 0 THEN
        IF NOT __ISVALIDREF(inoControl) THEN
            _varInfo := __VARINFO(inoControl);
            Messenger.Programming(_sb.Clear().Append('<#Invalid reference: #>').Append(_varInfo.Symbol).ToString()).Pin();
        ELSIF NOT __ISVALIDREF(inoConfig) THEN
            _varInfo := __VARINFO(inoConfig);
            Messenger.Programming(_sb.Clear().Append('<#Invalid reference: #>').Append(_varInfo.Symbol).ToString()).Pin();
        ELSIF NOT __ISVALIDREF(inoStatus) THEN
            _varInfo := __VARINFO(inoStatus);
            Messenger.Programming(_sb.Clear().Append('<#Invalid reference: #>').Append(_varInfo.Symbol).ToString()).Pin();
        ELSIF NOT inoStatus.ControllerInAuto THEN
            _varInfo := __VARINFO(inoStatus.ControllerInAuto);
            Messenger.Warning(_sb.Clear().Append('<#Tixon control system not in auto #>').Append(_varInfo.Symbol).ToString());
        ELSE
            IF NOT inoConfig.OutOfBoxSensorDisabled AND inoConfig.SeparatorHasWorkPosition THEN
                Messenger.Error(_sb.Clear()
                        .Append('<#Tixon has inconsistent configuration! (OutOfBoxSensorDisabled is not disabled instead of SeparatorHasWorkPosition is On!)#>')
                        .ToString()).Pin();
            ELSE
                IF NOT THIS^._errorMessage.Pinned THEN
                    _progress := _progress + 1;
                END_IF;
            END_IF;
        END_IF
    END_IF

    IF _progress = 1 THEN
        inoControl.SepareComponent := FALSE;
        _varInfo := __VARINFO(inoStatus.SeparatorHomePos);

        THIS^.Messenger.OnCondition(_infoTimer.Q AND NOT inoStatus.SeparatorHomePos)
            .Warning(_sb.Clear().Append('<#Waiting for #>').Append(_varInfo.Symbol).ToString());

        THIS^.Messenger.OnCondition(_infoTimer.Q AND inoStatus.ComponentOutOfBox AND NOT inoConfig.OutOfBoxSensorDisabled)
            .Error(_sb.Clear()
                .Append('<#Check component at the separator output. The component is probably stuck!.#>')
                .Append(_varInfo.Symbol)
                .ToString()).Pin();

        IF _infoTimer.Q AND inoStatus.ComponentOutOfBox and NOT inoConfig.OutOfBoxSensorDisabled THEN
            THIS^.ThrowWhen(_errorTimer.Q);
        ELSIF inoStatus.SeparatorHomePos AND NOT inoStatus.ComponentOutOfBox THEN
            _progress := _progress + 1;
            _timer(In := FALSE);
        END_IF;
    END_IF;

    IF _progress = 2 THEN
        Messenger.Debug('<#Waiting for component in  separator#>');
        _timer(IN := inoStatus.SeparatorPresent, Pt := inoConfig.TimeToComponentInSeparator);

        IF _timer.Q THEN
            _progress := _progress + 1;
            _timer(In := FALSE);
        END_IF
    END_IF;

    IF _progress = 3 THEN
        inoControl.SepareComponent := TRUE;
        Messenger.OnCondition(NOT inoConfig.OutOfBoxSensorDisabled).Debug('<#Waiting for component out of  separator#>');

        Messenger.OnCondition(inoConfig.OutOfBoxSensorDisabled AND inoConfig.SeparatorHasWorkPosition)
            .Warning('<#Waiting to separator to reach work position.#>');

        _timer(IN := inoStatus.SeparatorPresent, Pt := inoConfig.TimeToComponentOutSeparator);

        IF inoStatus.ComponentOutOfBox AND NOT inoConfig.OutOfBoxSensorDisabled THEN
            _progress := _progress + 1;
            _timer(In := FALSE);
        ELSIF inoConfig.OutOfBoxSensorDisabled AND inoConfig.SeparatorHasWorkPosition AND inoStatus.SeparatorWorkPos THEN
            _progress := _progress + 1;
            _timer(In := FALSE);
        ELSIF inoConfig.OutOfBoxSensorDisabled AND NOT inoConfig.SeparatorHasWorkPosition AND _timer.Q THEN
            _progress := _progress + 1;
            _timer(In := FALSE);
        ELSIF _timer.Q AND NOT inoConfig.OutOfBoxSensorDisabled THEN
            _progress := 1;
            _timer(In := FALSE);
        END_IF
    END_IF;

    IF _progress = 4 THEN
        _componentReady := TRUE;
        THIS^.DoneWhen(TRUE);
    END_IF;

    CallTimers(TRUE);
    THIS^.ThrowWhen(_errorTimer.Q);
END_IF

inoStatus.ComponentReady := _componentReady;

IF THIS^.Error AND NOT _errorMessage.Pinned THEN
    THIS^.Restore();
END_IF

PROPERTY PUBLIC ComponentReady : bool
GET
ComponentReady := _componentReady;
END_GET
END_PROPERTY

(*~
    <docu>
        <summary>
            Executes when task is aborted.
        </summary>
    </docu>
~*)
METHOD PROTECTED OnAbort
IF __ISVALIDREF(inoStatus) THEN
    THIS^.inoStatus.ActionDescription := '<#Separator task  was aborted.#>';
END_IF;
END_METHOD

(*~
    <docu>
        <summary>
            Executes when task reaches the ```Done``` state .
        </summary>
    </docu>
~*)
METHOD PROTECTED OnDone
IF __ISVALIDREF(inoStatus) THEN
    THIS^.inoStatus.ActionDescription := '<#Separator task  finished successfully.#>';
END_IF;

_progress := 0;

IF AutoRestore THEN
    Restore();
END_IF
END_METHOD

METHOD PROTECTED OnError
VAR
    description : STRING;
END_VAR
description := '<#Separator task finished with error.#>';
_componentReady := false;

IF __ISVALIDREF(inoStatus) THEN
    THIS^.inoStatus.ActionDescription := description;
END_IF;

THIS^._errorMessage.Error(_sb.Clear().Append(description).Append(' To restore acknowledge this alarm.').ToString()).Pin();
END_METHOD

